  MoveL 9409 to (-39.5, 44.85, 135.08) mm, rotated rx -180 ry 0 rz 180 deg; joints [-167.331, 69.156, -87.298, 166.691, 72.314, 4.11]
  Call Extruder(57.21099)
  MoveL 9410 to (-39.44, 44.66, 135.08) mm, rotated rx 180 ry 0 rz 180 deg; joints [-167.379, 69.148, -87.304, 166.74, 72.298, 4.098]
  MoveL 9411 to (-39.44, 44.66, 135.08) mm, rotated rx 180 ry 0 rz 180 deg; joints [-167.379, 69.148, -87.304, 166.74, 72.298, 4.098]
  Call Extruder(57.35863)
  MoveL 9412 to (-39.35, 44.42, 135.08) mm, rotated rx -180 ry 0 rz 180 deg; joints [-167.439, 69.136, -87.311, 166.802, 72.275, 4.084]
  MoveL 9413 to (-39.35, 44.42, 135.08) mm, rotated rx -180 ry 0 rz 180 deg; joints [-167.439, 69.136, -87.311, 166.802, 72.275, 4.084]
  Call Extruder(57.54097)
  MoveL 9414 to (-39.23, 44.13, 135.08) mm, rotated rx -180 ry 0 rz -180 deg; joints [-167.512, 69.122, -87.32, 166.876, 72.247, 4.066]
  MoveL 9415 to (-39.23, 44.13, 135.08) mm, rotated rx -180 ry 0 rz -180 deg; joints [-167.512, 69.122, -87.32, 166.876, 72.247, 4.066]
  Call Extruder(57.72406)
  MoveL 9416 to (-39.11, 43.83, 135.08) mm, rotated rx 180 ry 0 rz -180 deg; joints [-167.584, 69.107, -87.328, 166.951, 72.219, 4.049]
  MoveL 9417 to (-39.11, 43.83, 135.08) mm, rotated rx 180 ry 0 rz -180 deg; joints [-167.584, 69.107, -87.328, 166.951, 72.219, 4.049]
  Call Extruder(57.88175)
  MoveL 9418 to (-39, 43.58, 135.08) mm, rotated rx -180 ry 0 rz 180 deg; joints [-167.646, 69.094, -87.336, 167.014, 72.194, 4.034]
  MoveL 9419 to (-39, 43.58, 135.08) mm, rotated rx -180 ry 0 rz 180 deg; joints [-167.646, 69.094, -87.336, 167.014, 72.194, 4.034]
  Call Extruder(58.04004)
  MoveL 9420 to (-38.89, 43.33, 135.08) mm, rotated rx 180 ry 0 rz 180 deg; joints [-167.708, 69.081, -87.344, 167.078, 72.17, 4.019]
  MoveL 9421 to (-38.89, 43.33, 135.08) mm, rotated rx 180 ry 0 rz 180 deg; joints [-167.708, 69.081, -87.344, 167.078, 72.17, 4.019]
  Call Extruder(58.22206)
  MoveL 9422 to (-38.75, 43.06, 135.08) mm, rotated rx -180 ry 0 rz 180 deg; joints [-167.776, 69.065, -87.354, 167.147, 72.14, 4.003]
  MoveL 9423 to (-38.75, 43.06, 135.08) mm, rotated rx -180 ry 0 rz 180 deg; joints [-167.776, 69.065, -87.354, 167.147, 72.14, 4.003]
  Call Extruder(58.42862)
  MoveL 9424 to (-38.57, 42.75, 135.08) mm, rotated rx -180 ry 0 rz 180 deg; joints [-167.849, 69.046, -87.365, 167.222, 72.105, 3.986]
  MoveL 9425 to (-38.57, 42.75, 135.08) mm, rotated rx -180 ry 0 rz 180 deg; joints [-167.849, 69.046, -87.365, 167.222, 72.105, 3.986]
  Call Extruder(58.63595)
  MoveL 9426 to (-38.4, 42.45, 135.08) mm, rotated rx -180 ry 0 rz 180 deg; joints [-167.923, 69.027, -87.377, 167.296, 72.07, 3.97]
  MoveL 9427 to (-38.4, 42.45, 135.08) mm, rotated rx -180 ry 0 rz 180 deg; joints [-167.923, 69.027, -87.377, 167.296, 72.07, 3.97]
  Call Extruder(58.84406)
  MoveL 9428 to (-38.22, 42.15, 135.08) mm, rotated rx -180 ry 0 rz 180 deg; joints [-167.997, 69.007, -87.389, 167.371, 72.035, 3.953]
  MoveL 9429 to (-38.22, 42.15, 135.08) mm, rotated rx -180 ry 0 rz 180 deg; joints [-167.997, 69.007, -87.389, 167.371, 72.035, 3.953]
  Call Extruder(58.96178)
  MoveL 9430 to (-38.12, 41.98, 135.08) mm, rotated rx 180 ry 0 rz 180 deg; joints [-168.038, 68.997, -87.395, 167.414, 72.015, 3.944]
  MoveL 9431 to (-38.12, 41.98, 135.08) mm, rotated rx 180 ry 0 rz 180 deg; joints [-168.038, 68.997, -87.395, 167.414, 72.015, 3.944]
  Call Extruder(59.29462)
  MoveL 9432 to (-37.79, 41.52, 135.08) mm, rotated rx -180 ry 0 rz -180 deg; joints [-168.144, 68.962, -87.415, 167.521, 71.955, 3.922]
  MoveL 9433 to (-37.79, 41.52, 135.08) mm, rotated rx -180 ry 0 rz -180 deg; joints [-168.144, 68.962, -87.415, 167.521, 71.955, 3.922]
  Call Extruder(59.62865)
  MoveL 9434 to (-37.47, 41.07, 135.08) mm, rotated rx -180 ry 0 rz 180 deg; joints [-168.25, 68.929, -87.435, 167.629, 71.894, 3.899]
  MoveL 9435 to (-37.47, 41.07, 135.08) mm, rotated rx -180 ry 0 rz 180 deg; joints [-168.25, 68.929, -87.435, 167.629, 71.894, 3.899]
  Call Extruder(59.79624)
  MoveL 9436 to (-37.3, 40.85, 135.08) mm, rotated rx -180 ry 0 rz 180 deg; joints [-168.304, 68.912, -87.445, 167.683, 71.864, 3.888]
  Call Extruder(60.62555)
  MoveL 9437 to (-36.39, 39.81, 135.08) mm, rotated rx 180 ry 0 rz 180 deg; joints [-168.541, 68.821, -87.499, 167.922, 71.708, 3.842]
  Call Extruder(61.25663)
  MoveL 9438 to (-35.6, 39.11, 135.08) mm, rotated rx -180 ry 0 rz 180 deg; joints [-168.693, 68.746, -87.542, 168.074, 71.581, 3.818]
  MoveL 9439 to (-35.6, 39.11, 135.08) mm, rotated rx -180 ry 0 rz 180 deg; joints [-168.693, 68.746, -87.542, 168.074, 71.581, 3.818]
  Call Extruder(61.45419)
  MoveL 9440 to (-35.35, 38.9, 135.08) mm, rotated rx 180 ry 0 rz -180 deg; joints [-168.739, 68.722, -87.556, 168.12, 71.541, 3.811]
  Call Extruder(61.78821)
  MoveL 9441 to (-34.9, 38.57, 135.08) mm, rotated rx 180 ry 0 rz -180 deg; joints [-168.806, 68.68, -87.58, 168.186, 71.472, 3.803]
  MoveL 9442 to (-34.9, 38.57, 135.08) mm, rotated rx 180 ry 0 rz -180 deg; joints [-168.806, 68.68, -87.58, 168.186, 71.472, 3.803]
  Call Extruder(62.12104)
  MoveL 9443 to (-34.45, 38.24, 135.08) mm, rotated rx 180 ry 0 rz 180 deg; joints [-168.874, 68.638, -87.604, 168.253, 71.403, 3.794]
  MoveL 9444 to (-34.45, 38.24, 135.08) mm, rotated rx 180 ry 0 rz 180 deg; joints [-168.874, 68.638, -87.604, 168.253, 71.403, 3.794]
  Call Extruder(62.30029)
  MoveL 9445 to (-34.21, 38.07, 135.08) mm, rotated rx -180 ry 0 rz -180 deg; joints [-168.91, 68.615, -87.617, 168.288, 71.365, 3.79]
  MoveL 9446 to (-34.21, 38.07, 135.08) mm, rotated rx -180 ry 0 rz -180 deg; joints [-168.91, 68.615, -87.617, 168.288, 71.365, 3.79]
  Call Extruder(62.50840)
  MoveL 9447 to (-33.9, 37.89, 135.08) mm, rotated rx 180 ry 0 rz 180 deg; joints [-168.944, 68.587, -87.633, 168.32, 71.321, 3.788]
  MoveL 9448 to (-33.9, 37.89, 135.08) mm, rotated rx 180 ry 0 rz 180 deg; joints [-168.944, 68.587, -87.633, 168.32, 71.321, 3.788]
  Call Extruder(62.71573)
  MoveL 9449 to (-33.6, 37.71, 135.08) mm, rotated rx -180 ry 0 rz -180 deg; joints [-168.977, 68.559, -87.649, 168.352, 71.276, 3.786]
  MoveL 9450 to (-33.6, 37.71, 135.08) mm, rotated rx -180 ry 0 rz -180 deg; joints [-168.977, 68.559, -87.649, 168.352, 71.276, 3.786]
  Call Extruder(62.92229)
  MoveL 9451 to (-33.29, 37.54, 135.08) mm, rotated rx 180 ry 0 rz 180 deg; joints [-169.01, 68.531, -87.664, 168.384, 71.231, 3.784]
  MoveL 9452 to (-33.29, 37.54, 135.08) mm, rotated rx 180 ry 0 rz 180 deg; joints [-169.01, 68.531, -87.664, 168.384, 71.231, 3.784]
  Call Extruder(63.12806)
  MoveL 9453 to (-32.99, 37.36, 135.08) mm, rotated rx 180 ry 0 rz -180 deg; joints [-169.043, 68.504, -87.68, 168.416, 71.187, 3.782]
  MoveL 9454 to (-32.99, 37.36, 135.08) mm, rotated rx 180 ry 0 rz -180 deg; joints [-169.043, 68.504, -87.68, 168.416, 71.187, 3.782]
  Call Extruder(63.28636)
  MoveL 9455 to (-32.74, 37.26, 135.08) mm, rotated rx -180 ry 0 rz 180 deg; joints [-169.06, 68.481, -87.692, 168.432, 71.152, 3.783]
  MoveL 9456 to (-32.74, 37.26, 135.08) mm, rotated rx -180 ry 0 rz 180 deg; joints [-169.06, 68.481, -87.692, 168.432, 71.152, 3.783]
  Call Extruder(63.44406)
  MoveL 9457 to (-32.49, 37.15, 135.08) mm, rotated rx -180 ry 0 rz -180 deg; joints [-169.077, 68.459, -87.704, 168.447, 71.117, 3.785]
  MoveL 9458 to (-32.49, 37.15, 135.08) mm, rotated rx -180 ry 0 rz -180 deg; joints [-169.077, 68.459, -87.704, 168.447, 71.117, 3.785]
  Call Extruder(63.61415)
  MoveL 9459 to (-32.22, 37.04, 135.08) mm, rotated rx -180 ry 0 rz 180 deg; joints [-169.095, 68.435, -87.718, 168.463, 71.079, 3.787]
  MoveL 9460 to (-32.22, 37.04, 135.08) mm, rotated rx -180 ry 0 rz 180 deg; joints [-169.095, 68.435, -87.718, 168.463, 71.079, 3.787]
  Call Extruder(63.79648)
  MoveL 9461 to (-31.93, 36.91, 135.08) mm, rotated rx 180 ry 0 rz 180 deg; joints [-169.113, 68.409, -87.732, 168.48, 71.038, 3.789]
  MoveL 9462 to (-31.93, 36.91, 135.08) mm, rotated rx 180 ry 0 rz 180 deg; joints [-169.113, 68.409, -87.732, 168.48, 71.038, 3.789]
  Call Extruder(63.97805)
  MoveL 9463 to (-31.64, 36.79, 135.08) mm, rotated rx -180 ry 0 rz -180 deg; joints [-169.132, 68.383, -87.746, 168.497, 70.997, 3.791]
  MoveL 9464 to (-31.64, 36.79, 135.08) mm, rotated rx -180 ry 0 rz -180 deg; joints [-169.132, 68.383, -87.746, 168.497, 70.997, 3.791]
  Call Extruder(64.09151)
  MoveL 9465 to (-31.45, 36.73, 135.08) mm, rotated rx -180 ry 0 rz 180 deg; joints [-169.139, 68.366, -87.755, 168.503, 70.972, 3.794]
  MoveL 9466 to (-31.45, 36.73, 135.08) mm, rotated rx -180 ry 0 rz 180 deg; joints [-169.139, 68.366, -87.755, 168.503, 70.972, 3.794]
  Call Extruder(64.20453)
  MoveL 9467 to (-31.26, 36.67, 135.08) mm, rotated rx -180 ry 0 rz -180 deg; joints [-169.146, 68.35, -87.765, 168.509, 70.946, 3.797]
  MoveL 9468 to (-31.26, 36.67, 135.08) mm, rotated rx -180 ry 0 rz -180 deg; joints [-169.146, 68.35, -87.765, 168.509, 70.946, 3.797]
  Call Extruder(64.31709)
  MoveL 9469 to (-31.07, 36.61, 135.08) mm, rotated rx 180 ry 0 rz -180 deg; joints [-169.154, 68.333, -87.774, 168.515, 70.92, 3.8]
  MoveL 9470 to (-31.07, 36.61, 135.08) mm, rotated rx 180 ry 0 rz -180 deg; joints [-169.154, 68.333, -87.774, 168.515, 70.92, 3.8]
  Call Extruder(64.42922)
  MoveL 9471 to (-30.88, 36.55, 135.08) mm, rotated rx -180 ry 0 rz 180 deg; joints [-169.161, 68.316, -87.783, 168.521, 70.895, 3.803]
  MoveL 9472 to (-30.88, 36.55, 135.08) mm, rotated rx -180 ry 0 rz 180 deg; joints [-169.161, 68.316, -87.783, 168.521, 70.895, 3.803]
  Call Extruder(64.54090)
  MoveL 9473 to (-30.69, 36.49, 135.08) mm, rotated rx 180 ry 0 rz 180 deg; joints [-169.168, 68.3, -87.792, 168.527, 70.869, 3.806]
  MoveL 9474 to (-30.69, 36.49, 135.08) mm, rotated rx 180 ry 0 rz 180 deg; joints [-169.168, 68.3, -87.792, 168.527, 70.869, 3.806]
  Call Extruder(64.67197)
  MoveL 9475 to (-30.47, 36.42, 135.08) mm, rotated rx -180 ry 0 rz -180 deg; joints [-169.175, 68.28, -87.802, 168.532, 70.839, 3.809]
  MoveL 9476 to (-30.47, 36.42, 135.08) mm, rotated rx -180 ry 0 rz -180 deg; joints [-169.175, 68.28, -87.802, 168.532, 70.839, 3.809]
  Call Extruder(64.80248)
  MoveL 9477 to (-30.25, 36.35, 135.08) mm, rotated rx -180 ry 0 rz 180 deg; joints [-169.182, 68.26, -87.813, 168.538, 70.809, 3.813]
  MoveL 9478 to (-30.25, 36.35, 135.08) mm, rotated rx -180 ry 0 rz 180 deg; joints [-169.182, 68.26, -87.813, 168.538, 70.809, 3.813]
  Call Extruder(64.93242)
  MoveL 9479 to (-30.02, 36.28, 135.08) mm, rotated rx -180 ry 0 rz -180 deg; joints [-169.19, 68.241, -87.824, 168.543, 70.779, 3.817]
  MoveL 9480 to (-30.02, 36.28, 135.08) mm, rotated rx -180 ry 0 rz -180 deg; joints [-169.19, 68.241, -87.824, 168.543, 70.779, 3.817]
  Call Extruder(65.06180)
  MoveL 9481 to (-29.8, 36.22, 135.08) mm, rotated rx 180 ry 0 rz -180 deg; joints [-169.197, 68.221, -87.834, 168.549, 70.748, 3.821]
  MoveL 9482 to (-29.8, 36.22, 135.08) mm, rotated rx 180 ry 0 rz -180 deg; joints [-169.197, 68.221, -87.834, 168.549, 70.748, 3.821]
  Call Extruder(65.18377)
  MoveL 9483 to (-29.59, 36.16, 135.08) mm, rotated rx -180 ry 0 rz 180 deg; joints [-169.202, 68.202, -87.844, 168.552, 70.72, 3.826]
  MoveL 9484 to (-29.59, 36.16, 135.08) mm, rotated rx -180 ry 0 rz 180 deg; joints [-169.202, 68.202, -87.844, 168.552, 70.72, 3.826]
  Call Extruder(65.29861)
  MoveL 9485 to (-29.38, 36.12, 135.08) mm, rotated rx -180 ry 0 rz 180 deg; joints [-169.203, 68.185, -87.854, 168.551, 70.693, 3.831]
  MoveL 9486 to (-29.38, 36.12, 135.08) mm, rotated rx -180 ry 0 rz 180 deg; joints [-169.203, 68.185, -87.854, 168.551, 70.693, 3.831]
  Call Extruder(65.41301)
  MoveL 9487 to (-29.18, 36.07, 135.08) mm, rotated rx -180 ry 0 rz 180 deg; joints [-169.205, 68.167, -87.863, 168.551, 70.666, 3.836]
  MoveL 9488 to (-29.18, 36.07, 135.08) mm, rotated rx -180 ry 0 rz 180 deg; joints [-169.205, 68.167, -87.863, 168.551, 70.666, 3.836]
  Call Extruder(65.52695)
  MoveL 9489 to (-28.97, 36.03, 135.08) mm, rotated rx -180 ry 0 rz -180 deg; joints [-169.207, 68.149, -87.872, 168.551, 70.64, 3.841]
  MoveL 9490 to (-28.97, 36.03, 135.08) mm, rotated rx -180 ry 0 rz -180 deg; joints [-169.207, 68.149, -87.872, 168.551, 70.64, 3.841]
  Call Extruder(65.64044)
  MoveL 9491 to (-28.77, 35.98, 135.08) mm, rotated rx 180 ry 0 rz 180 deg; joints [-169.208, 68.131, -87.882, 168.551, 70.613, 3.846]
  MoveL 9492 to (-28.77, 35.98, 135.08) mm, rotated rx 180 ry 0 rz 180 deg; joints [-169.208, 68.131, -87.882, 168.551, 70.613, 3.846]
  Call Extruder(65.77772)
  MoveL 9493 to (-28.52, 35.93, 135.08) mm, rotated rx -180 ry 0 rz -180 deg; joints [-169.209, 68.11, -87.893, 168.549, 70.58, 3.853]
  MoveL 9494 to (-28.52, 35.93, 135.08) mm, rotated rx -180 ry 0 rz -180 deg; joints [-169.209, 68.11, -87.893, 168.549, 70.58, 3.853]
  Call Extruder(65.91440)
  MoveL 9495 to (-28.27, 35.88, 135.08) mm, rotated rx -180 ry 0 rz 180 deg; joints [-169.209, 68.088, -87.905, 168.547, 70.548, 3.86]
  MoveL 9496 to (-28.27, 35.88, 135.08) mm, rotated rx -180 ry 0 rz 180 deg; joints [-169.209, 68.088, -87.905, 168.547, 70.548, 3.86]
  Call Extruder(66.05046)
  MoveL 9497 to (-28.02, 35.83, 135.08) mm, rotated rx -180 ry 0 rz 180 deg; joints [-169.21, 68.066, -87.916, 168.546, 70.515, 3.866]
  MoveL 9498 to (-28.02, 35.83, 135.08) mm, rotated rx -180 ry 0 rz 180 deg; joints [-169.21, 68.066, -87.916, 168.546, 70.515, 3.866]
  Call Extruder(66.18591)
  MoveL 9499 to (-27.77, 35.78, 135.08) mm, rotated rx 180 ry 0 rz 180 deg; joints [-169.21, 68.044, -87.928, 168.544, 70.483, 3.873]
  MoveL 9500 to (-27.77, 35.78, 135.08) mm, rotated rx 180 ry 0 rz 180 deg; joints [-169.21, 68.044, -87.928, 168.544, 70.483, 3.873]
  Call Extruder(66.32075)
  MoveL 9501 to (-27.52, 35.73, 135.08) mm, rotated rx 180 ry 0 rz 180 deg; joints [-169.211, 68.023, -87.939, 168.543, 70.45, 3.88]
  MoveL 9502 to (-27.52, 35.73, 135.08) mm, rotated rx 180 ry 0 rz 180 deg; joints [-169.211, 68.023, -87.939, 168.543, 70.45, 3.88]
  Call Extruder(66.45498)
  MoveL 9503 to (-27.28, 35.68, 135.08) mm, rotated rx -180 ry 0 rz 180 deg; joints [-169.212, 68.001, -87.95, 168.541, 70.418, 3.887]
  MoveL 9504 to (-27.28, 35.68, 135.08) mm, rotated rx -180 ry 0 rz 180 deg; joints [-169.212, 68.001, -87.95, 168.541, 70.418, 3.887]
  Call Extruder(66.58860)
  MoveL 9505 to (-27.03, 35.63, 135.08) mm, rotated rx -180 ry 0 rz 180 deg; joints [-169.212, 67.979, -87.961, 168.539, 70.386, 3.893]
  MoveL 9506 to (-27.03, 35.63, 135.08) mm, rotated rx -180 ry 0 rz 180 deg; joints [-169.212, 67.979, -87.961, 168.539, 70.386, 3.893]
  Call Extruder(66.75070)
  MoveL 9507 to (-26.72, 35.59, 135.08) mm, rotated rx -180 ry 0 rz -180 deg; joints [-169.21, 67.953, -87.975, 168.533, 70.346, 3.903]
  MoveL 9508 to (-26.72, 35.59, 135.08) mm, rotated rx -180 ry 0 rz -180 deg; joints [-169.21, 67.953, -87.975, 168.533, 70.346, 3.903]
  Call Extruder(66.91207)
  MoveL 9509 to (-26.41, 35.54, 135.08) mm, rotated rx 180 ry 0 rz 180 deg; joints [-169.207, 67.926, -87.989, 168.527, 70.307, 3.913]
  MoveL 9510 to (-26.41, 35.54, 135.08) mm, rotated rx 180 ry 0 rz 180 deg; joints [-169.207, 67.926, -87.989, 168.527, 70.307, 3.913]
  Call Extruder(67.07271)
  MoveL 9511 to (-26.11, 35.49, 135.08) mm, rotated rx -180 ry 0 rz -180 deg; joints [-169.204, 67.899, -88.003, 168.521, 70.268, 3.922]
  MoveL 9512 to (-26.11, 35.49, 135.08) mm, rotated rx -180 ry 0 rz -180 deg; joints [-169.204, 67.899, -88.003, 168.521, 70.268, 3.922]
  Call Extruder(67.23263)
  MoveL 9513 to (-25.8, 35.44, 135.08) mm, rotated rx -180 ry 0 rz 180 deg; joints [-169.201, 67.873, -88.016, 168.515, 70.228, 3.932]
  MoveL 9514 to (-25.8, 35.44, 135.08) mm, rotated rx -180 ry 0 rz 180 deg; joints [-169.201, 67.873, -88.016, 168.515, 70.228, 3.932]
  Call Extruder(67.39181)
  MoveL 9515 to (-25.5, 35.39, 135.08) mm, rotated rx -180 ry 0 rz 180 deg; joints [-169.198, 67.846, -88.03, 168.51, 70.189, 3.941]
  MoveL 9516 to (-25.5, 35.39, 135.08) mm, rotated rx -180 ry 0 rz 180 deg; joints [-169.198, 67.846, -88.03, 168.51, 70.189, 3.941]
  Call Extruder(67.55027)
  MoveL 9517 to (-25.19, 35.34, 135.08) mm, rotated rx -180 ry 0 rz 180 deg; joints [-169.195, 67.819, -88.043, 168.503, 70.15, 3.951]
  MoveL 9518 to (-25.19, 35.34, 135.08) mm, rotated rx -180 ry 0 rz 180 deg; joints [-169.195, 67.819, -88.043, 168.503, 70.15, 3.951]
  Call Extruder(67.74915)
  MoveL 9519 to (-24.8, 35.3, 135.08) mm, rotated rx -180 ry 0 rz 180 deg; joints [-169.187, 67.786, -88.06, 168.491, 70.101, 3.965]
  MoveL 9520 to (-24.8, 35.3, 135.08) mm, rotated rx -180 ry 0 rz 180 deg; joints [-169.187, 67.786, -88.06, 168.491, 70.101, 3.965]
  Call Extruder(67.94716)
  MoveL 9521 to (-24.42, 35.25, 135.08) mm, rotated rx -180 ry 0 rz -180 deg; joints [-169.178, 67.752, -88.077, 168.478, 70.052, 3.978]
  MoveL 9522 to (-24.42, 35.25, 135.08) mm, rotated rx -180 ry 0 rz -180 deg; joints [-169.178, 67.752, -88.077, 168.478, 70.052, 3.978]
  Call Extruder(68.14430)
  MoveL 9523 to (-24.03, 35.21, 135.08) mm, rotated rx 180 ry 0 rz -180 deg; joints [-169.17, 67.718, -88.094, 168.466, 70.003, 3.992]
  MoveL 9524 to (-24.03, 35.21, 135.08) mm, rotated rx 180 ry 0 rz -180 deg; joints [-169.17, 67.718, -88.094, 168.466, 70.003, 3.992]
  Call Extruder(68.34057)
  MoveL 9525 to (-23.64, 35.16, 135.08) mm, rotated rx -180 ry 0 rz -180 deg; joints [-169.161, 67.684, -88.111, 168.453, 69.954, 4.006]
  MoveL 9526 to (-23.64, 35.16, 135.08) mm, rotated rx -180 ry 0 rz -180 deg; joints [-169.161, 67.684, -88.111, 168.453, 69.954, 4.006]
  Call Extruder(68.58626)
  MoveL 9527 to (-23.15, 35.11, 135.08) mm, rotated rx -180 ry 0 rz 180 deg; joints [-169.147, 67.642, -88.132, 168.433, 69.893, 4.025]
  MoveL 9528 to (-23.15, 35.11, 135.08) mm, rotated rx -180 ry 0 rz 180 deg; joints [-169.147, 67.642, -88.132, 168.433, 69.893, 4.025]
  Call Extruder(68.88099)
  MoveL 9529 to (-22.56, 35.07, 135.08) mm, rotated rx 180 ry 0 rz 180 deg; joints [-169.127, 67.591, -88.157, 168.406, 69.819, 4.048]
  MoveL 9530 to (-22.56, 35.07, 135.08) mm, rotated rx 180 ry 0 rz 180 deg; joints [-169.127, 67.591, -88.157, 168.406, 69.819, 4.048]
  Call Extruder(69.17439)
  MoveL 9531 to (-21.97, 35.02, 135.08) mm, rotated rx -180 ry 0 rz 180 deg; joints [-169.107, 67.539, -88.182, 168.379, 69.746, 4.072]
  MoveL 9532 to (-21.97, 35.02, 135.08) mm, rotated rx -180 ry 0 rz 180 deg; joints [-169.107, 67.539, -88.182, 168.379, 69.746, 4.072]
  Call Extruder(69.60772)
  MoveL 9533 to (-21.1, 34.98, 135.08) mm, rotated rx 180 ry 0 rz -180 deg; joints [-169.069, 67.463, -88.219, 168.331, 69.638, 4.11]
  MoveL 9534 to (-21.1, 34.98, 135.08) mm, rotated rx 180 ry 0 rz -180 deg; joints [-169.069, 67.463, -88.219, 168.331, 69.638, 4.11]
  Call Extruder(70.17988)
  MoveL 9535 to (-19.94, 34.93, 135.08) mm, rotated rx -180 ry 0 rz -180 deg; joints [-169.014, 67.362, -88.267, 168.261, 69.496, 4.163]
  MoveL 9536 to (-19.94, 34.93, 135.08) mm, rotated rx -180 ry 0 rz -180 deg; joints [-169.014, 67.362, -88.267, 168.261, 69.496, 4.163]
  Call Extruder(70.60771)
  MoveL 9537 to (-19.06, 34.91, 135.08) mm, rotated rx -180 ry 0 rz -180 deg; joints [-168.967, 67.286, -88.303, 168.202, 69.39, 4.205]
  Call Extruder(187.25639)
  MoveL 9538 to (219.06, 34.91, 135.08) mm, rotated rx 180 ry 0 rz -180 deg; joints [-30.588, 55.377, -90.527, 35.864, 119.71, 19.712]
  MoveL 9539 to (219.06, 34.91, 135.08) mm, rotated rx 180 ry 0 rz -180 deg; joints [-30.588, 55.377, -90.527, 35.864, 119.71, 19.712]
  Call Extruder(187.97196)
  MoveL 9540 to (220.52, 34.95, 135.08) mm, rotated rx -180 ry 0 rz 180 deg; joints [-30.009, 55.529, -90.53, 35.187, 119.782, 19.301]
  MoveL 9541 to (220.52, 34.95, 135.08) mm, rotated rx -180 ry 0 rz 180 deg; joints [-30.009, 55.529, -90.53, 35.187, 119.782, 19.301]
  Call Extruder(188.54670)
  MoveL 9542 to (221.68, 35, 135.08) mm, rotated rx 180 ry 0 rz 180 deg; joints [-29.572, 55.651, -90.532, 34.671, 119.826, 18.984]
  MoveL 9543 to (221.68, 35, 135.08) mm, rotated rx 180 ry 0 rz 180 deg; joints [-29.572, 55.651, -90.532, 34.671, 119.826, 18.984]
  Call Extruder(188.84009)
  MoveL 9544 to (222.27, 35.04, 135.08) mm, rotated rx -180 ry 0 rz 180 deg; joints [-29.371, 55.715, -90.532, 34.432, 119.839, 18.834]
  MoveL 9545 to (222.27, 35.04, 135.08) mm, rotated rx -180 ry 0 rz 180 deg; joints [-29.371, 55.715, -90.532, 34.432, 119.839, 18.834]
  Call Extruder(189.13482)
  MoveL 9546 to (222.86, 35.09, 135.08) mm, rotated rx -180 ry 0 rz 180 deg; joints [-29.173, 55.779, -90.533, 34.195, 119.851, 18.686]
  MoveL 9547 to (222.86, 35.09, 135.08) mm, rotated rx -180 ry 0 rz 180 deg; joints [-29.173, 55.779, -90.533, 34.195, 119.851, 18.686]
  Call Extruder(189.43087)
  MoveL 9548 to (223.45, 35.14, 135.08) mm, rotated rx -180 ry 0 rz -180 deg; joints [-28.978, 55.842, -90.534, 33.962, 119.861, 18.539]
  MoveL 9549 to (223.45, 35.14, 135.08) mm, rotated rx -180 ry 0 rz -180 deg; joints [-28.978, 55.842, -90.534, 33.962, 119.861, 18.539]
  Call Extruder(189.62715)
  MoveL 9550 to (223.84, 35.18, 135.08) mm, rotated rx 180 ry 0 rz 180 deg; joints [-28.862, 55.885, -90.534, 33.821, 119.863, 18.449]
  MoveL 9551 to (223.84, 35.18, 135.08) mm, rotated rx 180 ry 0 rz 180 deg; joints [-28.862, 55.885, -90.534, 33.821, 119.863, 18.449]
  Call Extruder(189.82429)
  MoveL 9552 to (224.22, 35.23, 135.08) mm, rotated rx 180 ry 0 rz 180 deg; joints [-28.747, 55.928, -90.534, 33.682, 119.864, 18.359]
  MoveL 9553 to (224.22, 35.23, 135.08) mm, rotated rx 180 ry 0 rz 180 deg; joints [-28.747, 55.928, -90.534, 33.682, 119.864, 18.359]
  Call Extruder(190.02230)
  MoveL 9554 to (224.61, 35.28, 135.08) mm, rotated rx 180 ry 0 rz -180 deg; joints [-28.633, 55.97, -90.534, 33.544, 119.864, 18.27]
  MoveL 9555 to (224.61, 35.28, 135.08) mm, rotated rx 180 ry 0 rz -180 deg; joints [-28.633, 55.97, -90.534, 33.544, 119.864, 18.27]
  Call Extruder(190.22117)
  MoveL 9556 to (225, 35.32, 135.08) mm, rotated rx -180 ry 0 rz 180 deg; joints [-28.52, 56.013, -90.535, 33.407, 119.864, 18.181]
  MoveL 9557 to (225, 35.32, 135.08) mm, rotated rx -180 ry 0 rz 180 deg; joints [-28.52, 56.013, -90.535, 33.407, 119.864, 18.181]
  Call Extruder(190.40025)
  MoveL 9558 to (225.34, 35.37, 135.08) mm, rotated rx -180 ry 0 rz 180 deg; joints [-28.425, 56.052, -90.535, 33.29, 119.862, 18.105]
  MoveL 9559 to (225.34, 35.37, 135.08) mm, rotated rx -180 ry 0 rz 180 deg; joints [-28.425, 56.052, -90.535, 33.29, 119.862, 18.105]
  Call Extruder(190.55944)
  MoveL 9560 to (225.65, 35.42, 135.08) mm, rotated rx -180 ry 0 rz 180 deg; joints [-28.346, 56.086, -90.535, 33.193, 119.857, 18.04]
  MoveL 9561 to (225.65, 35.42, 135.08) mm, rotated rx -180 ry 0 rz 180 deg; joints [-28.346, 56.086, -90.535, 33.193, 119.857, 18.04]
  Call Extruder(190.71935)
  MoveL 9562 to (225.96, 35.47, 135.08) mm, rotated rx 180 ry 0 rz 180 deg; joints [-28.267, 56.121, -90.535, 33.096, 119.853, 17.975]
  MoveL 9563 to (225.96, 35.47, 135.08) mm, rotated rx 180 ry 0 rz 180 deg; joints [-28.267, 56.121, -90.535, 33.096, 119.853, 17.975]
  Call Extruder(190.87999)
  MoveL 9564 to (226.26, 35.51, 135.08) mm, rotated rx -180 ry 0 rz 180 deg; joints [-28.19, 56.155, -90.535, 33, 119.848, 17.911]
  MoveL 9565 to (226.26, 35.51, 135.08) mm, rotated rx -180 ry 0 rz 180 deg; joints [-28.19, 56.155, -90.535, 33, 119.848, 17.911]
  Call Extruder(191.04136)
  MoveL 9566 to (226.57, 35.56, 135.08) mm, rotated rx 180 ry 0 rz 180 deg; joints [-28.112, 56.189, -90.535, 32.904, 119.843, 17.847]
  MoveL 9567 to (226.57, 35.56, 135.08) mm, rotated rx 180 ry 0 rz 180 deg; joints [-28.112, 56.189, -90.535, 32.904, 119.843, 17.847]
  Call Extruder(191.20345)
  MoveL 9568 to (226.87, 35.61, 135.08) mm, rotated rx 180 ry 0 rz 180 deg; joints [-28.036, 56.224, -90.535, 32.81, 119.837, 17.784]
  MoveL 9569 to (226.87, 35.61, 135.08) mm, rotated rx 180 ry 0 rz 180 deg; joints [-28.036, 56.224, -90.535, 32.81, 119.837, 17.784]
  Call Extruder(191.35165)
  MoveL 9570 to (227.15, 35.66, 135.08) mm, rotated rx -180 ry 0 rz -180 deg; joints [-27.971, 56.255, -90.535, 32.728, 119.83, 17.729]
  MoveL 9571 to (227.15, 35.66, 135.08) mm, rotated rx -180 ry 0 rz -180 deg; joints [-27.971, 56.255, -90.535, 32.728, 119.83, 17.729]
  Call Extruder(191.48588)
  MoveL 9572 to (227.4, 35.71, 135.08) mm, rotated rx -180 ry 0 rz 180 deg; joints [-27.915, 56.284, -90.534, 32.659, 119.823, 17.681]
  MoveL 9573 to (227.4, 35.71, 135.08) mm, rotated rx -180 ry 0 rz 180 deg; joints [-27.915, 56.284, -90.534, 32.659, 119.823, 17.681]
  Call Extruder(191.62072)
  MoveL 9574 to (227.65, 35.76, 135.08) mm, rotated rx -180 ry 0 rz 180 deg; joints [-27.861, 56.312, -90.534, 32.59, 119.815, 17.633]
  MoveL 9575 to (227.65, 35.76, 135.08) mm, rotated rx -180 ry 0 rz 180 deg; joints [-27.861, 56.312, -90.534, 32.59, 119.815, 17.633]
  Call Extruder(191.75618)
  MoveL 9576 to (227.9, 35.81, 135.08) mm, rotated rx -180 ry 0 rz 180 deg; joints [-27.807, 56.341, -90.534, 32.521, 119.808, 17.586]
  MoveL 9577 to (227.9, 35.81, 135.08) mm, rotated rx -180 ry 0 rz 180 deg; joints [-27.807, 56.341, -90.534, 32.521, 119.808, 17.586]
  Call Extruder(191.89224)
  MoveL 9578 to (228.15, 35.86, 135.08) mm, rotated rx -180 ry 0 rz 180 deg; joints [-27.753, 56.37, -90.534, 32.454, 119.8, 17.539]
  MoveL 9579 to (228.15, 35.86, 135.08) mm, rotated rx -180 ry 0 rz 180 deg; joints [-27.753, 56.37, -90.534, 32.454, 119.8, 17.539]
  Call Extruder(192.02891)
  MoveL 9580 to (228.4, 35.91, 135.08) mm, rotated rx -180 ry 0 rz -180 deg; joints [-27.699, 56.398, -90.534, 32.385, 119.792, 17.491]
  MoveL 9581 to (228.4, 35.91, 135.08) mm, rotated rx -180 ry 0 rz -180 deg; joints [-27.699, 56.398, -90.534, 32.385, 119.792, 17.491]
  Call Extruder(192.16620)
  MoveL 9582 to (228.65, 35.96, 135.08) mm, rotated rx 180 ry 0 rz 180 deg; joints [-27.646, 56.427, -90.534, 32.319, 119.783, 17.445]
  MoveL 9583 to (228.65, 35.96, 135.08) mm, rotated rx 180 ry 0 rz 180 deg; joints [-27.646, 56.427, -90.534, 32.319, 119.783, 17.445]
  Call Extruder(192.29187)
  MoveL 9584 to (228.87, 36, 135.08) mm, rotated rx -180 ry 0 rz -180 deg; joints [-27.599, 56.453, -90.533, 32.259, 119.775, 17.403]
  MoveL 9585 to (228.87, 36, 135.08) mm, rotated rx -180 ry 0 rz -180 deg; joints [-27.599, 56.453, -90.533, 32.259, 119.775, 17.403]
  Call Extruder(192.40582)
  MoveL 9586 to (229.08, 36.05, 135.08) mm, rotated rx -180 ry 0 rz 180 deg; joints [-27.559, 56.476, -90.533, 32.207, 119.767, 17.366]
  MoveL 9587 to (229.08, 36.05, 135.08) mm, rotated rx -180 ry 0 rz 180 deg; joints [-27.559, 56.476, -90.533, 32.207, 119.767, 17.366]
  Call Extruder(192.52022)
  MoveL 9588 to (229.28, 36.09, 135.08) mm, rotated rx 180 ry 0 rz 180 deg; joints [-27.518, 56.5, -90.533, 32.156, 119.759, 17.33]
  MoveL 9589 to (229.28, 36.09, 135.08) mm, rotated rx 180 ry 0 rz 180 deg; joints [-27.518, 56.5, -90.533, 32.156, 119.759, 17.33]
  Call Extruder(192.63507)
  MoveL 9590 to (229.48, 36.14, 135.08) mm, rotated rx -180 ry 0 rz -180 deg; joints [-27.479, 56.524, -90.533, 32.105, 119.75, 17.293]
  MoveL 9591 to (229.48, 36.14, 135.08) mm, rotated rx -180 ry 0 rz -180 deg; joints [-27.479, 56.524, -90.533, 32.105, 119.75, 17.293]
  Call Extruder(192.75038)
  MoveL 9592 to (229.69, 36.18, 135.08) mm, rotated rx 180 ry 0 rz 180 deg; joints [-27.439, 56.547, -90.532, 32.054, 119.742, 17.257]
  MoveL 9593 to (229.69, 36.18, 135.08) mm, rotated rx 180 ry 0 rz 180 deg; joints [-27.439, 56.547, -90.532, 32.054, 119.742, 17.257]
  Call Extruder(192.82364)
  MoveL 9594 to (229.82, 36.22, 135.08) mm, rotated rx -180 ry 0 rz 180 deg; joints [-27.421, 56.562, -90.532, 32.029, 119.734, 17.238]
  MoveL 9595 to (229.82, 36.22, 135.08) mm, rotated rx -180 ry 0 rz 180 deg; joints [-27.421, 56.562, -90.532, 32.029, 119.734, 17.238]
  Call Extruder(192.95114)
  MoveL 9596 to (230.03, 36.29, 135.08) mm, rotated rx -180 ry 0 rz 180 deg; joints [-27.39, 56.589, -90.532, 31.987, 119.721, 17.205]
  MoveL 9597 to (230.03, 36.29, 135.08) mm, rotated rx -180 ry 0 rz 180 deg; joints [-27.39, 56.589, -90.532, 31.987, 119.721, 17.205]
  Call Extruder(193.07920)
  MoveL 9598 to (230.25, 36.35, 135.08) mm, rotated rx -180 ry 0 rz 180 deg; joints [-27.36, 56.615, -90.532, 31.946, 119.707, 17.172]
  MoveL 9599 to (230.25, 36.35, 135.08) mm, rotated rx -180 ry 0 rz 180 deg; joints [-27.36, 56.615, -90.532, 31.946, 119.707, 17.172]
  Call Extruder(193.20780)
  MoveL 9600 to (230.48, 36.42, 135.08) mm, rotated rx 180 ry 0 rz -180 deg; joints [-27.329, 56.642, -90.531, 31.904, 119.693, 17.139]
  MoveL 9601 to (230.48, 36.42, 135.08) mm, rotated rx 180 ry 0 rz -180 deg; joints [-27.329, 56.642, -90.531, 31.904, 119.693, 17.139]
  Call Extruder(193.33694)
  MoveL 9602 to (230.7, 36.49, 135.08) mm, rotated rx -180 ry 0 rz -180 deg; joints [-27.299, 56.668, -90.531, 31.863, 119.679, 17.106]
  MoveL 9603 to (230.7, 36.49, 135.08) mm, rotated rx -180 ry 0 rz -180 deg; joints [-27.299, 56.668, -90.531, 31.863, 119.679, 17.106]
  Call Extruder(193.44884)
  MoveL 9604 to (230.88, 36.55, 135.08) mm, rotated rx 180 ry 0 rz -180 deg; joints [-27.276, 56.691, -90.53, 31.831, 119.667, 17.08]
  MoveL 9605 to (230.88, 36.55, 135.08) mm, rotated rx 180 ry 0 rz -180 deg; joints [-27.276, 56.691, -90.53, 31.831, 119.667, 17.08]
  Call Extruder(193.56118)
  MoveL 9606 to (231.07, 36.61, 135.08) mm, rotated rx 180 ry 0 rz 180 deg; joints [-27.253, 56.714, -90.53, 31.798, 119.654, 17.053]
  MoveL 9607 to (231.07, 36.61, 135.08) mm, rotated rx 180 ry 0 rz 180 deg; joints [-27.253, 56.714, -90.53, 31.798, 119.654, 17.053]
  Call Extruder(193.67397)
  MoveL 9608 to (231.26, 36.67, 135.08) mm, rotated rx -180 ry 0 rz -180 deg; joints [-27.231, 56.736, -90.53, 31.767, 119.64, 17.027]
  MoveL 9609 to (231.26, 36.67, 135.08) mm, rotated rx -180 ry 0 rz -180 deg; joints [-27.231, 56.736, -90.53, 31.767, 119.64, 17.027]
  Call Extruder(193.78720)
  MoveL 9610 to (231.45, 36.73, 135.08) mm, rotated rx 180 ry 0 rz 180 deg; joints [-27.208, 56.759, -90.529, 31.735, 119.627, 17]
  MoveL 9611 to (231.45, 36.73, 135.08) mm, rotated rx 180 ry 0 rz 180 deg; joints [-27.208, 56.759, -90.529, 31.735, 119.627, 17]
  Call Extruder(193.90088)
  MoveL 9612 to (231.64, 36.79, 135.08) mm, rotated rx -180 ry 0 rz -180 deg; joints [-27.185, 56.782, -90.529, 31.703, 119.614, 16.974]
  MoveL 9613 to (231.64, 36.79, 135.08) mm, rotated rx -180 ry 0 rz -180 deg; joints [-27.185, 56.782, -90.529, 31.703, 119.614, 16.974]
  Call Extruder(194.08284)
  MoveL 9614 to (231.93, 36.91, 135.08) mm, rotated rx -180 ry 0 rz -180 deg; joints [-27.167, 56.819, -90.528, 31.672, 119.588, 16.941]
  MoveL 9615 to (231.93, 36.91, 135.08) mm, rotated rx -180 ry 0 rz -180 deg; joints [-27.167, 56.819, -90.528, 31.672, 119.588, 16.941]
  Call Extruder(194.26556)
  MoveL 9616 to (232.22, 37.04, 135.08) mm, rotated rx 180 ry 0 rz 180 deg; joints [-27.149, 56.855, -90.527, 31.641, 119.561, 16.909]
  MoveL 9617 to (232.22, 37.04, 135.08) mm, rotated rx 180 ry 0 rz 180 deg; joints [-27.149, 56.855, -90.527, 31.641, 119.561, 16.909]
  Call Extruder(194.43598)
  MoveL 9618 to (232.49, 37.15, 135.08) mm, rotated rx -180 ry 0 rz -180 deg; joints [-27.133, 56.889, -90.527, 31.613, 119.536, 16.88]
  MoveL 9619 to (232.49, 37.15, 135.08) mm, rotated rx -180 ry 0 rz -180 deg; joints [-27.133, 56.889, -90.527, 31.613, 119.536, 16.88]
  Call Extruder(194.59398)
  MoveL 9620 to (232.74, 37.26, 135.08) mm, rotated rx 180 ry 0 rz 180 deg; joints [-27.121, 56.921, -90.526, 31.59, 119.513, 16.854]
  MoveL 9621 to (232.74, 37.26, 135.08) mm, rotated rx 180 ry 0 rz 180 deg; joints [-27.121, 56.921, -90.526, 31.59, 119.513, 16.854]
  Call Extruder(194.75258)
  MoveL 9622 to (232.99, 37.36, 135.08) mm, rotated rx 180 ry 0 rz 180 deg; joints [-27.108, 56.952, -90.525, 31.566, 119.489, 16.827]
  MoveL 9623 to (232.99, 37.36, 135.08) mm, rotated rx 180 ry 0 rz 180 deg; joints [-27.108, 56.952, -90.525, 31.566, 119.489, 16.827]
  Call Extruder(194.95874)
  MoveL 9624 to (233.29, 37.54, 135.08) mm, rotated rx 180 ry 0 rz 180 deg; joints [-27.12, 56.993, -90.524, 31.567, 119.45, 16.809]
  MoveL 9625 to (233.29, 37.54, 135.08) mm, rotated rx 180 ry 0 rz 180 deg; joints [-27.12, 56.993, -90.524, 31.567, 119.45, 16.809]
  Call Extruder(195.16569)
  MoveL 9626 to (233.6, 37.71, 135.08) mm, rotated rx -180 ry 0 rz 180 deg; joints [-27.132, 57.034, -90.523, 31.568, 119.411, 16.79]
  MoveL 9627 to (233.6, 37.71, 135.08) mm, rotated rx -180 ry 0 rz 180 deg; joints [-27.132, 57.034, -90.523, 31.568, 119.411, 16.79]
  Call Extruder(195.37341)
  MoveL 9628 to (233.9, 37.89, 135.08) mm, rotated rx 180 ry 0 rz 180 deg; joints [-27.144, 57.074, -90.522, 31.569, 119.372, 16.772]
  MoveL 9629 to (233.9, 37.89, 135.08) mm, rotated rx 180 ry 0 rz 180 deg; joints [-27.144, 57.074, -90.522, 31.569, 119.372, 16.772]
  Call Extruder(195.58192)
  MoveL 9630 to (234.21, 38.07, 135.08) mm, rotated rx -180 ry 0 rz 180 deg; joints [-27.156, 57.115, -90.521, 31.57, 119.333, 16.753]
  MoveL 9631 to (234.21, 38.07, 135.08) mm, rotated rx -180 ry 0 rz 180 deg; joints [-27.156, 57.115, -90.521, 31.57, 119.333, 16.753]
  Call Extruder(195.76146)
  MoveL 9632 to (234.45, 38.24, 135.08) mm, rotated rx -180 ry 0 rz 180 deg; joints [-27.187, 57.149, -90.52, 31.593, 119.294, 16.748]
  MoveL 9633 to (234.45, 38.24, 135.08) mm, rotated rx -180 ry 0 rz 180 deg; joints [-27.187, 57.149, -90.52, 31.593, 119.294, 16.748]
  Call Extruder(196.09487)
  MoveL 9634 to (234.9, 38.57, 135.08) mm, rotated rx 180 ry 0 rz 180 deg; joints [-27.245, 57.213, -90.518, 31.638, 119.221, 16.74]
  MoveL 9635 to (234.9, 38.57, 135.08) mm, rotated rx 180 ry 0 rz 180 deg; joints [-27.245, 57.213, -90.518, 31.638, 119.221, 16.74]
  Call Extruder(196.42947)
  MoveL 9636 to (235.35, 38.9, 135.08) mm, rotated rx 180 ry 0 rz 180 deg; joints [-27.302, 57.277, -90.516, 31.681, 119.148, 16.731]
  Call Extruder(197.25742)
  MoveL 9637 to (236.39, 39.81, 135.08) mm, rotated rx -180 ry 0 rz -180 deg; joints [-27.525, 57.431, -90.511, 31.879, 118.948, 16.753]
  Call Extruder(198.08537)
  MoveL 9638 to (237.3, 40.85, 135.08) mm, rotated rx -180 ry 0 rz 180 deg; joints [-27.851, 57.58, -90.505, 32.19, 118.723, 16.832]
  Call Extruder(198.25267)
  MoveL 9639 to (237.47, 41.07, 135.08) mm, rotated rx -180 ry 0 rz 180 deg; joints [-27.932, 57.608, -90.504, 32.269, 118.675, 16.856]
  MoveL 9640 to (237.47, 41.07, 135.08) mm, rotated rx -180 ry 0 rz 180 deg; joints [-27.932, 57.608, -90.504, 32.269, 118.675, 16.856]
  Call Extruder(198.58609)
  MoveL 9641 to (237.79, 41.52, 135.08) mm, rotated rx -180 ry 0 rz -180 deg; joints [-28.091, 57.666, -90.501, 32.425, 118.578, 16.902]
  MoveL 9642 to (237.79, 41.52, 135.08) mm, rotated rx -180 ry 0 rz -180 deg; joints [-28.091, 57.666, -90.501, 32.425, 118.578, 16.902]
  Call Extruder(198.91833)
  MoveL 9643 to (238.12, 41.97, 135.08) mm, rotated rx -180 ry 0 rz 180 deg; joints [-28.249, 57.724, -90.498, 32.579, 118.481, 16.947]
  MoveL 9644 to (238.12, 41.97, 135.08) mm, rotated rx -180 ry 0 rz 180 deg; joints [-28.249, 57.724, -90.498, 32.579, 118.481, 16.947]
  Call Extruder(199.03601)
  MoveL 9645 to (238.22, 42.15, 135.08) mm, rotated rx 180 ry 0 rz 180 deg; joints [-28.315, 57.743, -90.497, 32.646, 118.444, 16.97]
  MoveL 9646 to (238.22, 42.15, 135.08) mm, rotated rx 180 ry 0 rz 180 deg; joints [-28.315, 57.743, -90.497, 32.646, 118.444, 16.97]
  Call Extruder(199.24373)
  MoveL 9647 to (238.4, 42.45, 135.08) mm, rotated rx 180 ry 0 rz 180 deg; joints [-28.434, 57.777, -90.496, 32.764, 118.38, 17.009]
  MoveL 9648 to (238.4, 42.45, 135.08) mm, rotated rx 180 ry 0 rz 180 deg; joints [-28.434, 57.777, -90.496, 32.764, 118.38, 17.009]
  Call Extruder(199.45067)
  MoveL 9649 to (238.57, 42.75, 135.08) mm, rotated rx 180 ry 0 rz -180 deg; joints [-28.552, 57.811, -90.494, 32.882, 118.315, 17.048]
  MoveL 9650 to (238.57, 42.75, 135.08) mm, rotated rx 180 ry 0 rz -180 deg; joints [-28.552, 57.811, -90.494, 32.882, 118.315, 17.048]
  Call Extruder(199.65683)
  MoveL 9651 to (238.75, 43.06, 135.08) mm, rotated rx -180 ry 0 rz 180 deg; joints [-28.669, 57.845, -90.493, 32.998, 118.251, 17.086]
  MoveL 9652 to (238.75, 43.06, 135.08) mm, rotated rx -180 ry 0 rz 180 deg; joints [-28.669, 57.845, -90.493, 32.998, 118.251, 17.086]
  Call Extruder(199.83852)
  MoveL 9653 to (238.89, 43.34, 135.08) mm, rotated rx 180 ry 0 rz 180 deg; joints [-28.78, 57.875, -90.491, 33.11, 118.192, 17.124]
  MoveL 9654 to (238.89, 43.34, 135.08) mm, rotated rx 180 ry 0 rz 180 deg; joints [-28.78, 57.875, -90.491, 33.11, 118.192, 17.124]
  Call Extruder(199.99654)
  MoveL 9655 to (239, 43.58, 135.08) mm, rotated rx -180 ry 0 rz 180 deg; joints [-28.886, 57.899, -90.49, 33.217, 118.139, 17.162]
  MoveL 9656 to (239, 43.58, 135.08) mm, rotated rx -180 ry 0 rz 180 deg; joints [-28.886, 57.899, -90.49, 33.217, 118.139, 17.162]
  Call Extruder(200.15395)
  MoveL 9657 to (239.11, 43.83, 135.08) mm, rotated rx 180 ry 0 rz -180 deg; joints [-28.991, 57.924, -90.488, 33.324, 118.087, 17.2]
  MoveL 9658 to (239.11, 43.83, 135.08) mm, rotated rx 180 ry 0 rz -180 deg; joints [-28.991, 57.924, -90.488, 33.324, 118.087, 17.2]
  Call Extruder(200.33666)
  MoveL 9659 to (239.22, 44.12, 135.08) mm, rotated rx -180 ry 0 rz 180 deg; joints [-29.116, 57.952, -90.487, 33.45, 118.025, 17.245]
  MoveL 9660 to (239.22, 44.12, 135.08) mm, rotated rx -180 ry 0 rz 180 deg; joints [-29.116, 57.952, -90.487, 33.45, 118.025, 17.245]
  Call Extruder(200.51862)
  MoveL 9661 to (239.35, 44.42, 135.08) mm, rotated rx -180 ry 0 rz -180 deg; joints [-29.24, 57.98, -90.485, 33.575, 117.963, 17.289]
  MoveL 9662 to (239.35, 44.42, 135.08) mm, rotated rx -180 ry 0 rz -180 deg; joints [-29.24, 57.98, -90.485, 33.575, 117.963, 17.289]
  Call Extruder(200.66595)
  MoveL 9663 to (239.44, 44.66, 135.08) mm, rotated rx 180 ry 0 rz -180 deg; joints [-29.343, 58.003, -90.484, 33.68, 117.913, 17.326]
  MoveL 9664 to (239.44, 44.66, 135.08) mm, rotated rx 180 ry 0 rz -180 deg; joints [-29.343, 58.003, -90.484, 33.68, 117.913, 17.326]
  Call Extruder(200.77919)
  MoveL 9665 to (239.5, 44.85, 135.08) mm, rotated rx -180 ry 0 rz 180 deg; joints [-29.428, 58.019, -90.483, 33.766, 117.873, 17.358]
  MoveL 9666 to (239.5, 44.85, 135.08) mm, rotated rx -180 ry 0 rz 180 deg; joints [-29.428, 58.019, -90.483, 33.766, 117.873, 17.358]
  Call Extruder(200.89198)
  MoveL 9667 to (239.56, 45.03, 135.08) mm, rotated rx -180 ry 0 rz -180 deg; joints [-29.512, 58.036, -90.482, 33.852, 117.833, 17.389]
  MoveL 9668 to (239.56, 45.03, 135.08) mm, rotated rx -180 ry 0 rz -180 deg; joints [-29.512, 58.036, -90.482, 33.852, 117.833, 17.389]
  Call Extruder(201.00432)
  MoveL 9669 to (239.62, 45.22, 135.08) mm, rotated rx -180 ry 0 rz 180 deg; joints [-29.596, 58.053, -90.481, 33.937, 117.794, 17.42]
  MoveL 9670 to (239.62, 45.22, 135.08) mm, rotated rx -180 ry 0 rz 180 deg; joints [-29.596, 58.053, -90.481, 33.937, 117.794, 17.42]
  Call Extruder(201.11622)
  MoveL 9671 to (239.68, 45.41, 135.08) mm, rotated rx 180 ry 0 rz 180 deg; joints [-29.679, 58.069, -90.481, 34.022, 117.754, 17.451]
  MoveL 9672 to (239.68, 45.41, 135.08) mm, rotated rx 180 ry 0 rz 180 deg; joints [-29.679, 58.069, -90.481, 34.022, 117.754, 17.451]
  Call Extruder(201.23762)
  MoveL 9673 to (239.75, 45.62, 135.08) mm, rotated rx 180 ry 0 rz 180 deg; joints [-29.77, 58.087, -90.479, 34.115, 117.711, 17.485]
  MoveL 9674 to (239.75, 45.62, 135.08) mm, rotated rx 180 ry 0 rz 180 deg; joints [-29.77, 58.087, -90.479, 34.115, 117.711, 17.485]
  Call Extruder(201.36842)
  MoveL 9675 to (239.82, 45.84, 135.08) mm, rotated rx 180 ry 0 rz 180 deg; joints [-29.871, 58.107, -90.478, 34.217, 117.664, 17.522]
  MoveL 9676 to (239.82, 45.84, 135.08) mm, rotated rx 180 ry 0 rz 180 deg; joints [-29.871, 58.107, -90.478, 34.217, 117.664, 17.522]
  Call Extruder(201.49864)
  MoveL 9677 to (239.88, 46.06, 135.08) mm, rotated rx 180 ry 0 rz 180 deg; joints [-29.97, 58.126, -90.477, 34.318, 117.617, 17.559]
  MoveL 9678 to (239.88, 46.06, 135.08) mm, rotated rx 180 ry 0 rz 180 deg; joints [-29.97, 58.126, -90.477, 34.318, 117.617, 17.559]
  Call Extruder(201.62830)
  MoveL 9679 to (239.95, 46.29, 135.08) mm, rotated rx -180 ry 0 rz -180 deg; joints [-30.069, 58.145, -90.476, 34.418, 117.57, 17.595]
  MoveL 9680 to (239.95, 46.29, 135.08) mm, rotated rx -180 ry 0 rz -180 deg; joints [-30.069, 58.145, -90.476, 34.418, 117.57, 17.595]
  Call Extruder(201.75740)
  MoveL 9681 to (240.02, 46.51, 135.08) mm, rotated rx -180 ry 0 rz 180 deg; joints [-30.168, 58.165, -90.475, 34.519, 117.523, 17.631]
  MoveL 9682 to (240.02, 46.51, 135.08) mm, rotated rx -180 ry 0 rz 180 deg; joints [-30.168, 58.165, -90.475, 34.519, 117.523, 17.631]
  Call Extruder(201.87246)
  MoveL 9683 to (240.06, 46.72, 135.08) mm, rotated rx -180 ry 0 rz 180 deg; joints [-30.263, 58.181, -90.474, 34.616, 117.48, 17.668]
  MoveL 9684 to (240.06, 46.72, 135.08) mm, rotated rx -180 ry 0 rz 180 deg; joints [-30.263, 58.181, -90.474, 34.616, 117.48, 17.668]
  Call Extruder(201.98706)
  MoveL 9685 to (240.11, 46.92, 135.08) mm, rotated rx -180 ry 0 rz 180 deg; joints [-30.358, 58.197, -90.473, 34.713, 117.437, 17.704]
  MoveL 9686 to (240.11, 46.92, 135.08) mm, rotated rx -180 ry 0 rz 180 deg; joints [-30.358, 58.197, -90.473, 34.713, 117.437, 17.704]
  Call Extruder(202.10121)
  MoveL 9687 to (240.15, 47.12, 135.08) mm, rotated rx 180 ry 0 rz 180 deg; joints [-30.453, 58.213, -90.472, 34.809, 117.395, 17.739]
  MoveL 9688 to (240.15, 47.12, 135.08) mm, rotated rx 180 ry 0 rz 180 deg; joints [-30.453, 58.213, -90.472, 34.809, 117.395, 17.739]
  Call Extruder(202.21491)
  MoveL 9689 to (240.2, 47.33, 135.08) mm, rotated rx 180 ry 0 rz 180 deg; joints [-30.548, 58.229, -90.471, 34.906, 117.352, 17.775]
  MoveL 9690 to (240.2, 47.33, 135.08) mm, rotated rx 180 ry 0 rz 180 deg; joints [-30.548, 58.229, -90.471, 34.906, 117.352, 17.775]
  Call Extruder(202.34032)
  MoveL 9691 to (240.24, 47.55, 135.08) mm, rotated rx 180 ry 0 rz 180 deg; joints [-30.653, 58.247, -90.47, 35.013, 117.304, 17.815]
  MoveL 9692 to (240.24, 47.55, 135.08) mm, rotated rx 180 ry 0 rz 180 deg; joints [-30.653, 58.247, -90.47, 35.013, 117.304, 17.815]
  Call Extruder(202.47730)
  MoveL 9693 to (240.29, 47.8, 135.08) mm, rotated rx -180 ry 0 rz 180 deg; joints [-30.768, 58.266, -90.469, 35.13, 117.252, 17.858]
  MoveL 9694 to (240.29, 47.8, 135.08) mm, rotated rx -180 ry 0 rz 180 deg; joints [-30.768, 58.266, -90.469, 35.13, 117.252, 17.858]
  Call Extruder(202.61366)
  MoveL 9695 to (240.34, 48.05, 135.08) mm, rotated rx -180 ry 0 rz 180 deg; joints [-30.884, 58.285, -90.467, 35.248, 117.2, 17.901]
  MoveL 9696 to (240.34, 48.05, 135.08) mm, rotated rx -180 ry 0 rz 180 deg; joints [-30.884, 58.285, -90.467, 35.248, 117.2, 17.901]
  Call Extruder(202.74942)
  MoveL 9697 to (240.39, 48.3, 135.08) mm, rotated rx 180 ry 0 rz 180 deg; joints [-30.999, 58.305, -90.466, 35.365, 117.147, 17.944]
  MoveL 9698 to (240.39, 48.3, 135.08) mm, rotated rx 180 ry 0 rz 180 deg; joints [-30.999, 58.305, -90.466, 35.365, 117.147, 17.944]
  Call Extruder(202.88457)
  MoveL 9699 to (240.44, 48.55, 135.08) mm, rotated rx 180 ry 0 rz 180 deg; joints [-31.114, 58.324, -90.465, 35.482, 117.095, 17.987]
  MoveL 9700 to (240.44, 48.55, 135.08) mm, rotated rx 180 ry 0 rz 180 deg; joints [-31.114, 58.324, -90.465, 35.482, 117.095, 17.987]
  Call Extruder(203.01910)
  MoveL 9701 to (240.49, 48.8, 135.08) mm, rotated rx -180 ry 0 rz 180 deg; joints [-31.228, 58.343, -90.464, 35.598, 117.043, 18.029]
  MoveL 9702 to (240.49, 48.8, 135.08) mm, rotated rx -180 ry 0 rz 180 deg; joints [-31.228, 58.343, -90.464, 35.598, 117.043, 18.029]
  Call Extruder(203.15303)
  MoveL 9703 to (240.54, 49.05, 135.08) mm, rotated rx -180 ry 0 rz 180 deg; joints [-31.342, 58.363, -90.462, 35.713, 116.991, 18.071]
  MoveL 9704 to (240.54, 49.05, 135.08) mm, rotated rx -180 ry 0 rz 180 deg; joints [-31.342, 58.363, -90.462, 35.713, 116.991, 18.071]
  Call Extruder(203.30090)
  MoveL 9705 to (240.59, 49.33, 135.08) mm, rotated rx 180 ry 0 rz 180 deg; joints [-31.47, 58.384, -90.461, 35.843, 116.933, 18.118]
  MoveL 9706 to (240.59, 49.33, 135.08) mm, rotated rx 180 ry 0 rz 180 deg; joints [-31.47, 58.384, -90.461, 35.843, 116.933, 18.118]
  Call Extruder(203.46264)
  MoveL 9707 to (240.64, 49.63, 135.08) mm, rotated rx 180 ry 0 rz 180 deg; joints [-31.612, 58.407, -90.46, 35.987, 116.869, 18.17]
  MoveL 9708 to (240.64, 49.63, 135.08) mm, rotated rx 180 ry 0 rz 180 deg; joints [-31.612, 58.407, -90.46, 35.987, 116.869, 18.17]
  Call Extruder(203.62365)
  MoveL 9709 to (240.69, 49.94, 135.08) mm, rotated rx -180 ry 0 rz 180 deg; joints [-31.755, 58.429, -90.458, 36.132, 116.805, 18.223]
  MoveL 9710 to (240.69, 49.94, 135.08) mm, rotated rx -180 ry 0 rz 180 deg; joints [-31.755, 58.429, -90.458, 36.132, 116.805, 18.223]
  Call Extruder(203.78394)
  MoveL 9711 to (240.74, 50.24, 135.08) mm, rotated rx -180 ry 0 rz 180 deg; joints [-31.895, 58.452, -90.456, 36.274, 116.741, 18.274]
  MoveL 9712 to (240.74, 50.24, 135.08) mm, rotated rx -180 ry 0 rz 180 deg; joints [-31.895, 58.452, -90.456, 36.274, 116.741, 18.274]
  Call Extruder(203.94350)
  MoveL 9713 to (240.78, 50.55, 135.08) mm, rotated rx -180 ry 0 rz 180 deg; joints [-32.036, 58.475, -90.455, 36.416, 116.677, 18.325]
  MoveL 9714 to (240.78, 50.55, 135.08) mm, rotated rx -180 ry 0 rz 180 deg; joints [-32.036, 58.475, -90.455, 36.416, 116.677, 18.325]
  Call Extruder(204.10233)
  MoveL 9715 to (240.83, 50.86, 135.08) mm, rotated rx -180 ry 0 rz 180 deg; joints [-32.176, 58.498, -90.453, 36.558, 116.613, 18.375]
  MoveL 9716 to (240.83, 50.86, 135.08) mm, rotated rx -180 ry 0 rz 180 deg; joints [-32.176, 58.498, -90.453, 36.558, 116.613, 18.375]
  Call Extruder(204.28100)
  MoveL 9717 to (240.88, 51.2, 135.08) mm, rotated rx 180 ry 0 rz 180 deg; joints [-32.337, 58.524, -90.451, 36.72, 116.541, 18.433]
  MoveL 9718 to (240.88, 51.2, 135.08) mm, rotated rx 180 ry 0 rz 180 deg; joints [-32.337, 58.524, -90.451, 36.72, 116.541, 18.433]
  Call Extruder(204.47945)
  MoveL 9719 to (240.93, 51.59, 135.08) mm, rotated rx 180 ry 0 rz 180 deg; joints [-32.518, 58.551, -90.449, 36.903, 116.46, 18.499]
  MoveL 9720 to (240.93, 51.59, 135.08) mm, rotated rx 180 ry 0 rz 180 deg; joints [-32.518, 58.551, -90.449, 36.903, 116.46, 18.499]
  Call Extruder(204.67702)
  MoveL 9721 to (240.97, 51.98, 135.08) mm, rotated rx -180 ry 0 rz 180 deg; joints [-32.697, 58.579, -90.447, 37.084, 116.379, 18.563]
  MoveL 9722 to (240.97, 51.98, 135.08) mm, rotated rx -180 ry 0 rz 180 deg; joints [-32.697, 58.579, -90.447, 37.084, 116.379, 18.563]
  Call Extruder(204.87373)
  MoveL 9723 to (241.02, 52.37, 135.08) mm, rotated rx -180 ry 0 rz -180 deg; joints [-32.876, 58.607, -90.445, 37.264, 116.298, 18.627]
  MoveL 9724 to (241.02, 52.37, 135.08) mm, rotated rx -180 ry 0 rz -180 deg; joints [-32.876, 58.607, -90.445, 37.264, 116.298, 18.627]
  Call Extruder(205.06957)
  MoveL 9725 to (241.06, 52.75, 135.08) mm, rotated rx 180 ry 0 rz 180 deg; joints [-33.055, 58.635, -90.443, 37.444, 116.217, 18.69]
  MoveL 9726 to (241.06, 52.75, 135.08) mm, rotated rx 180 ry 0 rz 180 deg; joints [-33.055, 58.635, -90.443, 37.444, 116.217, 18.69]
  Call Extruder(205.36500)
  MoveL 9727 to (241.11, 53.34, 135.08) mm, rotated rx 180 ry 0 rz -180 deg; joints [-33.331, 58.676, -90.44, 37.722, 116.093, 18.789]
  MoveL 9728 to (241.11, 53.34, 135.08) mm, rotated rx 180 ry 0 rz -180 deg; joints [-33.331, 58.676, -90.44, 37.722, 116.093, 18.789]
  Call Extruder(205.65911)
  MoveL 9729 to (241.15, 53.93, 135.08) mm, rotated rx -180 ry 0 rz 180 deg; joints [-33.606, 58.717, -90.437, 37.998, 115.97, 18.886]
  MoveL 9730 to (241.15, 53.93, 135.08) mm, rotated rx -180 ry 0 rz 180 deg; joints [-33.606, 58.717, -90.437, 37.998, 115.97, 18.886]
  Call Extruder(205.95189)
  MoveL 9731 to (241.2, 54.52, 135.08) mm, rotated rx 180 ry 0 rz 180 deg; joints [-33.878, 58.758, -90.434, 38.272, 115.846, 18.981]
  MoveL 9732 to (241.2, 54.52, 135.08) mm, rotated rx 180 ry 0 rz 180 deg; joints [-33.878, 58.758, -90.434, 38.272, 115.846, 18.981]
  Call Extruder(206.52534)
  MoveL 9733 to (241.25, 55.68, 135.08) mm, rotated rx 180 ry 0 rz 180 deg; joints [-34.425, 58.836, -90.428, 38.82, 115.602, 19.171]
  MoveL 9734 to (241.25, 55.68, 135.08) mm, rotated rx 180 ry 0 rz 180 deg; joints [-34.425, 58.836, -90.428, 38.82, 115.602, 19.171]
  Call Extruder(207.23917)
  MoveL 9735 to (241.29, 57.14, 135.08) mm, rotated rx 180 ry 0 rz 180 deg; joints [-35.104, 58.932, -90.42, 39.498, 115.297, 19.404]
  Call Extruder(249.30405)
  MoveL 9736 to (241.29, 142.86, 135.08) mm, rotated rx -180 ry 0 rz 180 deg; joints [-60.361, 65.64, -88.988, 62.418, 101.303, 20.565]
  Call Extruder(249.73248)
  MoveL 9737 to (241.27, 143.74, 135.08) mm, rotated rx 180 ry 0 rz 180 deg; joints [-60.516, 65.711, -88.962, 62.548, 101.204, 20.507]
  MoveL 9738 to (241.27, 143.74, 135.08) mm, rotated rx 180 ry 0 rz 180 deg; joints [-60.516, 65.711, -88.962, 62.548, 101.204, 20.507]
  Call Extruder(250.30594)
  MoveL 9739 to (241.22, 144.9, 135.08) mm, rotated rx -180 ry 0 rz 180 deg; joints [-60.726, 65.804, -88.928, 62.728, 101.071, 20.43]
  MoveL 9740 to (241.22, 144.9, 135.08) mm, rotated rx -180 ry 0 rz 180 deg; joints [-60.726, 65.804, -88.928, 62.728, 101.071, 20.43]
  Call Extruder(250.74027)
  MoveL 9741 to (241.18, 145.77, 135.08) mm, rotated rx 180 ry 0 rz 180 deg; joints [-60.887, 65.873, -88.901, 62.865, 100.972, 20.373]
  MoveL 9742 to (241.18, 145.77, 135.08) mm, rotated rx 180 ry 0 rz 180 deg; joints [-60.887, 65.873, -88.901, 62.865, 100.972, 20.373]
  Call Extruder(251.03438)
  MoveL 9743 to (241.13, 146.36, 135.08) mm, rotated rx 180 ry 0 rz -180 deg; joints [-61, 65.919, -88.884, 62.961, 100.904, 20.336]
  MoveL 9744 to (241.13, 146.36, 135.08) mm, rotated rx 180 ry 0 rz -180 deg; joints [-61, 65.919, -88.884, 62.961, 100.904, 20.336]
  Call Extruder(251.32982)
  MoveL 9745 to (241.09, 146.95, 135.08) mm, rotated rx -180 ry 0 rz 180 deg; joints [-61.111, 65.964, -88.866, 63.056, 100.836, 20.299]
  MoveL 9746 to (241.09, 146.95, 135.08) mm, rotated rx -180 ry 0 rz 180 deg; joints [-61.111, 65.964, -88.866, 63.056, 100.836, 20.299]
  Call Extruder(251.57607)
  MoveL 9747 to (241.04, 147.44, 135.08) mm, rotated rx -180 ry 0 rz 180 deg; joints [-61.205, 66.002, -88.852, 63.137, 100.78, 20.268]
  MoveL 9748 to (241.04, 147.44, 135.08) mm, rotated rx -180 ry 0 rz 180 deg; joints [-61.205, 66.002, -88.852, 63.137, 100.78, 20.268]
  Call Extruder(251.77278)
  MoveL 9749 to (240.99, 147.83, 135.08) mm, rotated rx -180 ry 0 rz -180 deg; joints [-61.282, 66.032, -88.84, 63.204, 100.735, 20.245]
  MoveL 9750 to (240.99, 147.83, 135.08) mm, rotated rx -180 ry 0 rz -180 deg; joints [-61.282, 66.032, -88.84, 63.204, 100.735, 20.245]
  Call Extruder(251.97035)
  MoveL 9751 to (240.95, 148.22, 135.08) mm, rotated rx -180 ry 0 rz 180 deg; joints [-61.359, 66.061, -88.829, 63.27, 100.69, 20.221]
  MoveL 9752 to (240.95, 148.22, 135.08) mm, rotated rx -180 ry 0 rz 180 deg; joints [-61.359, 66.061, -88.829, 63.27, 100.69, 20.221]
  Call Extruder(252.16879)
  MoveL 9753 to (240.9, 148.6, 135.08) mm, rotated rx -180 ry 0 rz 180 deg; joints [-61.436, 66.09, -88.817, 63.337, 100.645, 20.197]
  MoveL 9754 to (240.9, 148.6, 135.08) mm, rotated rx -180 ry 0 rz 180 deg; joints [-61.436, 66.09, -88.817, 63.337, 100.645, 20.197]
  Call Extruder(252.36810)
  MoveL 9755 to (240.86, 148.99, 135.08) mm, rotated rx -180 ry 0 rz 180 deg; joints [-61.512, 66.12, -88.806, 63.403, 100.601, 20.173]
  MoveL 9756 to (240.86, 148.99, 135.08) mm, rotated rx -180 ry 0 rz 180 deg; joints [-61.512, 66.12, -88.806, 63.403, 100.601, 20.173]
  Call Extruder(252.52693)
  MoveL 9757 to (240.81, 149.3, 135.08) mm, rotated rx 180 ry 0 rz 180 deg; joints [-61.575, 66.142, -88.797, 63.458, 100.564, 20.156]
  MoveL 9758 to (240.81, 149.3, 135.08) mm, rotated rx 180 ry 0 rz 180 deg; joints [-61.575, 66.142, -88.797, 63.458, 100.564, 20.156]
  Call Extruder(252.68649)
  MoveL 9759 to (240.76, 149.6, 135.08) mm, rotated rx -180 ry 0 rz 180 deg; joints [-61.639, 66.165, -88.788, 63.513, 100.528, 20.138]
  MoveL 9760 to (240.76, 149.6, 135.08) mm, rotated rx -180 ry 0 rz 180 deg; joints [-61.639, 66.165, -88.788, 63.513, 100.528, 20.138]
  Call Extruder(252.84678)
  MoveL 9761 to (240.71, 149.91, 135.08) mm, rotated rx 180 ry 0 rz 180 deg; joints [-61.702, 66.188, -88.779, 63.568, 100.493, 20.12]
  MoveL 9762 to (240.71, 149.91, 135.08) mm, rotated rx 180 ry 0 rz 180 deg; joints [-61.702, 66.188, -88.779, 63.568, 100.493, 20.12]
  Call Extruder(253.00780)
  MoveL 9763 to (240.66, 150.21, 135.08) mm, rotated rx -180 ry 0 rz 180 deg; joints [-61.765, 66.21, -88.77, 63.623, 100.457, 20.102]
  MoveL 9764 to (240.66, 150.21, 135.08) mm, rotated rx -180 ry 0 rz 180 deg; joints [-61.765, 66.21, -88.77, 63.623, 100.457, 20.102]
  Call Extruder(253.16954)
  MoveL 9765 to (240.61, 150.52, 135.08) mm, rotated rx -180 ry 0 rz 180 deg; joints [-61.828, 66.233, -88.76, 63.678, 100.421, 20.084]
  MoveL 9766 to (240.61, 150.52, 135.08) mm, rotated rx -180 ry 0 rz 180 deg; joints [-61.828, 66.233, -88.76, 63.678, 100.421, 20.084]
  Call Extruder(253.33202)
  MoveL 9767 to (240.56, 150.83, 135.08) mm, rotated rx -180 ry 0 rz 180 deg; joints [-61.891, 66.256, -88.751, 63.733, 100.385, 20.066]
  MoveL 9768 to (240.56, 150.83, 135.08) mm, rotated rx -180 ry 0 rz 180 deg; joints [-61.891, 66.256, -88.751, 63.733, 100.385, 20.066]
  Call Extruder(253.46594)
  MoveL 9769 to (240.52, 151.08, 135.08) mm, rotated rx 180 ry 0 rz -180 deg; joints [-61.944, 66.274, -88.744, 63.78, 100.356, 20.052]
  MoveL 9770 to (240.52, 151.08, 135.08) mm, rotated rx 180 ry 0 rz -180 deg; joints [-61.944, 66.274, -88.744, 63.78, 100.356, 20.052]
  Call Extruder(253.60048)
  MoveL 9771 to (240.47, 151.32, 135.08) mm, rotated rx 180 ry 0 rz -180 deg; joints [-61.998, 66.292, -88.737, 63.827, 100.326, 20.038]
  MoveL 9772 to (240.47, 151.32, 135.08) mm, rotated rx 180 ry 0 rz -180 deg; joints [-61.998, 66.292, -88.737, 63.827, 100.326, 20.038]
  Call Extruder(253.73563)
  MoveL 9773 to (240.42, 151.57, 135.08) mm, rotated rx 180 ry 0 rz 180 deg; joints [-62.052, 66.31, -88.729, 63.875, 100.297, 20.024]
  MoveL 9774 to (240.42, 151.57, 135.08) mm, rotated rx 180 ry 0 rz 180 deg; joints [-62.052, 66.31, -88.729, 63.875, 100.297, 20.024]
  Call Extruder(253.87138)
  MoveL 9775 to (240.37, 151.82, 135.08) mm, rotated rx 180 ry 0 rz -180 deg; joints [-62.105, 66.328, -88.722, 63.922, 100.267, 20.01]
  MoveL 9776 to (240.37, 151.82, 135.08) mm, rotated rx 180 ry 0 rz -180 deg; joints [-62.105, 66.328, -88.722, 63.922, 100.267, 20.01]
  Call Extruder(254.00775)
  MoveL 9777 to (240.32, 152.07, 135.08) mm, rotated rx -180 ry 0 rz 180 deg; joints [-62.159, 66.346, -88.715, 63.969, 100.238, 19.996]
  MoveL 9778 to (240.32, 152.07, 135.08) mm, rotated rx -180 ry 0 rz 180 deg; joints [-62.159, 66.346, -88.715, 63.969, 100.238, 19.996]
  Call Extruder(254.14473)
  MoveL 9779 to (240.27, 152.32, 135.08) mm, rotated rx 180 ry 0 rz 180 deg; joints [-62.212, 66.364, -88.707, 64.015, 100.208, 19.982]
  MoveL 9780 to (240.27, 152.32, 135.08) mm, rotated rx 180 ry 0 rz 180 deg; joints [-62.212, 66.364, -88.707, 64.015, 100.208, 19.982]
  Call Extruder(254.28232)
  MoveL 9781 to (240.22, 152.57, 135.08) mm, rotated rx -180 ry 0 rz 180 deg; joints [-62.265, 66.382, -88.7, 64.062, 100.179, 19.968]
  MoveL 9782 to (240.22, 152.57, 135.08) mm, rotated rx -180 ry 0 rz 180 deg; joints [-62.265, 66.382, -88.7, 64.062, 100.179, 19.968]
  Call Extruder(254.39601)
  MoveL 9783 to (240.17, 152.77, 135.08) mm, rotated rx -180 ry 0 rz 180 deg; joints [-62.31, 66.397, -88.694, 64.101, 100.155, 19.956]
  MoveL 9784 to (240.17, 152.77, 135.08) mm, rotated rx -180 ry 0 rz 180 deg; joints [-62.31, 66.397, -88.694, 64.101, 100.155, 19.956]
  Call Extruder(254.51016)
  MoveL 9785 to (240.13, 152.98, 135.08) mm, rotated rx -180 ry 0 rz 180 deg; joints [-62.355, 66.411, -88.688, 64.14, 100.13, 19.945]
  MoveL 9786 to (240.13, 152.98, 135.08) mm, rotated rx -180 ry 0 rz 180 deg; joints [-62.355, 66.411, -88.688, 64.14, 100.13, 19.945]
  Call Extruder(254.62477)
  MoveL 9787 to (240.08, 153.18, 135.08) mm, rotated rx -180 ry 0 rz 180 deg; joints [-62.399, 66.426, -88.682, 64.18, 100.106, 19.934]
  MoveL 9788 to (240.08, 153.18, 135.08) mm, rotated rx -180 ry 0 rz 180 deg; joints [-62.399, 66.426, -88.682, 64.18, 100.106, 19.934]
  Call Extruder(254.73982)
  MoveL 9789 to (240.04, 153.39, 135.08) mm, rotated rx -180 ry 0 rz -180 deg; joints [-62.444, 66.441, -88.676, 64.219, 100.082, 19.922]
  MoveL 9790 to (240.04, 153.39, 135.08) mm, rotated rx -180 ry 0 rz -180 deg; joints [-62.444, 66.441, -88.676, 64.219, 100.082, 19.922]
  Call Extruder(254.86204)
  MoveL 9791 to (239.98, 153.6, 135.08) mm, rotated rx -180 ry 0 rz 180 deg; joints [-62.493, 66.456, -88.67, 64.262, 100.056, 19.911]
  MoveL 9792 to (239.98, 153.6, 135.08) mm, rotated rx -180 ry 0 rz 180 deg; joints [-62.493, 66.456, -88.67, 64.262, 100.056, 19.911]
  Call Extruder(254.99170)
  MoveL 9793 to (239.92, 153.82, 135.08) mm, rotated rx -180 ry 0 rz 180 deg; joints [-62.547, 66.471, -88.663, 64.31, 100.028, 19.9]
  MoveL 9794 to (239.92, 153.82, 135.08) mm, rotated rx -180 ry 0 rz 180 deg; joints [-62.547, 66.471, -88.663, 64.31, 100.028, 19.9]
  Call Extruder(255.12193)
  MoveL 9795 to (239.85, 154.05, 135.08) mm, rotated rx -180 ry 0 rz 180 deg; joints [-62.601, 66.486, -88.657, 64.358, 100.001, 19.889]
  MoveL 9796 to (239.85, 154.05, 135.08) mm, rotated rx -180 ry 0 rz 180 deg; joints [-62.601, 66.486, -88.657, 64.358, 100.001, 19.889]
  Call Extruder(255.25272)
  MoveL 9797 to (239.78, 154.27, 135.08) mm, rotated rx 180 ry 0 rz -180 deg; joints [-62.654, 66.501, -88.651, 64.406, 99.973, 19.878]
  MoveL 9798 to (239.78, 154.27, 135.08) mm, rotated rx 180 ry 0 rz -180 deg; joints [-62.654, 66.501, -88.651, 64.406, 99.973, 19.878]
  Call Extruder(255.38407)
  MoveL 9799 to (239.71, 154.49, 135.08) mm, rotated rx -180 ry 0 rz 180 deg; joints [-62.708, 66.517, -88.644, 64.454, 99.945, 19.867]
  MoveL 9800 to (239.71, 154.49, 135.08) mm, rotated rx -180 ry 0 rz 180 deg; joints [-62.708, 66.517, -88.644, 64.454, 99.945, 19.867]
  Call Extruder(255.49598)
  MoveL 9801 to (239.65, 154.68, 135.08) mm, rotated rx -180 ry 0 rz 180 deg; joints [-62.754, 66.529, -88.639, 64.496, 99.922, 19.859]
  MoveL 9802 to (239.65, 154.68, 135.08) mm, rotated rx -180 ry 0 rz 180 deg; joints [-62.754, 66.529, -88.639, 64.496, 99.922, 19.859]
  Call Extruder(255.60832)
  MoveL 9803 to (239.59, 154.87, 135.08) mm, rotated rx -180 ry 0 rz 180 deg; joints [-62.801, 66.542, -88.633, 64.537, 99.899, 19.85]
  MoveL 9804 to (239.59, 154.87, 135.08) mm, rotated rx -180 ry 0 rz 180 deg; joints [-62.801, 66.542, -88.633, 64.537, 99.899, 19.85]
  Call Extruder(255.72111)
  MoveL 9805 to (239.53, 155.06, 135.08) mm, rotated rx -180 ry 0 rz 180 deg; joints [-62.847, 66.555, -88.628, 64.578, 99.875, 19.841]
  MoveL 9806 to (239.53, 155.06, 135.08) mm, rotated rx -180 ry 0 rz 180 deg; joints [-62.847, 66.555, -88.628, 64.578, 99.875, 19.841]
  Call Extruder(255.83435)
  MoveL 9807 to (239.47, 155.25, 135.08) mm, rotated rx -180 ry 0 rz 180 deg; joints [-62.893, 66.567, -88.623, 64.62, 99.852, 19.832]
  MoveL 9808 to (239.47, 155.25, 135.08) mm, rotated rx -180 ry 0 rz 180 deg; joints [-62.893, 66.567, -88.623, 64.62, 99.852, 19.832]
  Call Extruder(255.94803)
  MoveL 9809 to (239.41, 155.44, 135.08) mm, rotated rx -180 ry 0 rz -180 deg; joints [-62.939, 66.58, -88.617, 64.661, 99.828, 19.823]
  MoveL 9810 to (239.41, 155.44, 135.08) mm, rotated rx -180 ry 0 rz -180 deg; joints [-62.939, 66.58, -88.617, 64.661, 99.828, 19.823]
  Call Extruder(256.12998)
  MoveL 9811 to (239.29, 155.73, 135.08) mm, rotated rx -180 ry 0 rz 180 deg; joints [-63.018, 66.599, -88.61, 64.732, 99.79, 19.811]
  MoveL 9812 to (239.29, 155.73, 135.08) mm, rotated rx -180 ry 0 rz 180 deg; joints [-63.018, 66.599, -88.61, 64.732, 99.79, 19.811]
  Call Extruder(256.31270)
  MoveL 9813 to (239.16, 156.02, 135.08) mm, rotated rx -180 ry 0 rz 180 deg; joints [-63.097, 66.617, -88.602, 64.803, 99.752, 19.8]
  MoveL 9814 to (239.16, 156.02, 135.08) mm, rotated rx -180 ry 0 rz 180 deg; joints [-63.097, 66.617, -88.602, 64.803, 99.752, 19.8]
  Call Extruder(256.48312)
  MoveL 9815 to (239.05, 156.29, 135.08) mm, rotated rx 180 ry 0 rz 180 deg; joints [-63.17, 66.635, -88.594, 64.869, 99.717, 19.789]
  MoveL 9816 to (239.05, 156.29, 135.08) mm, rotated rx 180 ry 0 rz 180 deg; joints [-63.17, 66.635, -88.594, 64.869, 99.717, 19.789]
  Call Extruder(256.64113)
  MoveL 9817 to (238.94, 156.54, 135.08) mm, rotated rx -180 ry 0 rz -180 deg; joints [-63.238, 66.65, -88.588, 64.93, 99.685, 19.779]
  MoveL 9818 to (238.94, 156.54, 135.08) mm, rotated rx -180 ry 0 rz -180 deg; joints [-63.238, 66.65, -88.588, 64.93, 99.685, 19.779]
  Call Extruder(256.79975)
  MoveL 9819 to (238.84, 156.79, 135.08) mm, rotated rx -180 ry 0 rz -180 deg; joints [-63.306, 66.666, -88.581, 64.992, 99.652, 19.769]
  MoveL 9820 to (238.84, 156.79, 135.08) mm, rotated rx -180 ry 0 rz -180 deg; joints [-63.306, 66.666, -88.581, 64.992, 99.652, 19.769]
  Call Extruder(257.00592)
  MoveL 9821 to (238.66, 157.09, 135.08) mm, rotated rx 180 ry 0 rz 180 deg; joints [-63.401, 66.684, -88.573, 65.079, 99.609, 19.762]
  MoveL 9822 to (238.66, 157.09, 135.08) mm, rotated rx 180 ry 0 rz 180 deg; joints [-63.401, 66.684, -88.573, 65.079, 99.609, 19.762]
  Call Extruder(257.21287)
  MoveL 9823 to (238.49, 157.4, 135.08) mm, rotated rx 180 ry 0 rz 180 deg; joints [-63.497, 66.701, -88.566, 65.166, 99.566, 19.754]
  MoveL 9824 to (238.49, 157.4, 135.08) mm, rotated rx 180 ry 0 rz 180 deg; joints [-63.497, 66.701, -88.566, 65.166, 99.566, 19.754]
  Call Extruder(257.42059)
  MoveL 9825 to (238.31, 157.7, 135.08) mm, rotated rx 180 ry 0 rz 180 deg; joints [-63.592, 66.719, -88.558, 65.253, 99.524, 19.746]
  MoveL 9826 to (238.31, 157.7, 135.08) mm, rotated rx 180 ry 0 rz 180 deg; joints [-63.592, 66.719, -88.558, 65.253, 99.524, 19.746]
  Call Extruder(257.62910)
  MoveL 9827 to (238.14, 158.01, 135.08) mm, rotated rx -180 ry 0 rz -180 deg; joints [-63.687, 66.736, -88.551, 65.34, 99.481, 19.738]
  MoveL 9828 to (238.14, 158.01, 135.08) mm, rotated rx -180 ry 0 rz -180 deg; joints [-63.687, 66.736, -88.551, 65.34, 99.481, 19.738]
  Call Extruder(257.80864)
  MoveL 9829 to (237.96, 158.25, 135.08) mm, rotated rx -180 ry 0 rz 180 deg; joints [-63.774, 66.749, -88.545, 65.42, 99.444, 19.734]
  MoveL 9830 to (237.96, 158.25, 135.08) mm, rotated rx -180 ry 0 rz 180 deg; joints [-63.774, 66.749, -88.545, 65.42, 99.444, 19.734]
  Call Extruder(258.14205)
  MoveL 9831 to (237.63, 158.7, 135.08) mm, rotated rx -180 ry 0 rz -180 deg; joints [-63.934, 66.772, -88.535, 65.568, 99.376, 19.728]
  MoveL 9832 to (237.63, 158.7, 135.08) mm, rotated rx -180 ry 0 rz -180 deg; joints [-63.934, 66.772, -88.535, 65.568, 99.376, 19.728]
  Call Extruder(258.47664)
  MoveL 9833 to (237.3, 159.15, 135.08) mm, rotated rx 180 ry 0 rz 180 deg; joints [-64.094, 66.796, -88.525, 65.715, 99.308, 19.722]
  Call Extruder(259.30463)
  MoveL 9834 to (236.39, 160.19, 135.08) mm, rotated rx -180 ry 0 rz -180 deg; joints [-64.505, 66.845, -88.503, 66.097, 99.141, 19.72]
  Call Extruder(260.13252)
  MoveL 9835 to (235.35, 161.1, 135.08) mm, rotated rx -180 ry 0 rz 180 deg; joints [-64.933, 66.879, -88.488, 66.498, 98.977, 19.738]
  Call Extruder(260.29983)
  MoveL 9836 to (235.13, 161.27, 135.08) mm, rotated rx -180 ry 0 rz 180 deg; joints [-65.021, 66.884, -88.486, 66.581, 98.944, 19.745]
  MoveL 9837 to (235.13, 161.27, 135.08) mm, rotated rx -180 ry 0 rz 180 deg; joints [-65.021, 66.884, -88.486, 66.581, 98.944, 19.745]
  Call Extruder(260.63326)
  MoveL 9838 to (234.68, 161.59, 135.08) mm, rotated rx 180 ry 0 rz 180 deg; joints [-65.197, 66.893, -88.482, 66.747, 98.879, 19.758]
  MoveL 9839 to (234.68, 161.59, 135.08) mm, rotated rx 180 ry 0 rz 180 deg; joints [-65.197, 66.893, -88.482, 66.747, 98.879, 19.758]
  Call Extruder(260.96550)
  MoveL 9840 to (234.23, 161.92, 135.08) mm, rotated rx 180 ry 0 rz -180 deg; joints [-65.374, 66.903, -88.478, 66.912, 98.814, 19.771]
  MoveL 9841 to (234.23, 161.92, 135.08) mm, rotated rx 180 ry 0 rz -180 deg; joints [-65.374, 66.903, -88.478, 66.912, 98.814, 19.771]
  Call Extruder(261.08316)
  MoveL 9842 to (234.05, 162.02, 135.08) mm, rotated rx -180 ry 0 rz 180 deg; joints [-65.437, 66.905, -88.477, 66.972, 98.791, 19.778]
  MoveL 9843 to (234.05, 162.02, 135.08) mm, rotated rx -180 ry 0 rz 180 deg; joints [-65.437, 66.905, -88.477, 66.972, 98.791, 19.778]
  Call Extruder(261.29090)
  MoveL 9844 to (233.75, 162.2, 135.08) mm, rotated rx 180 ry 0 rz 180 deg; joints [-65.549, 66.908, -88.475, 67.079, 98.752, 19.79]
  MoveL 9845 to (233.75, 162.2, 135.08) mm, rotated rx 180 ry 0 rz 180 deg; joints [-65.549, 66.908, -88.475, 67.079, 98.752, 19.79]
  Call Extruder(261.49785)
  MoveL 9846 to (233.45, 162.37, 135.08) mm, rotated rx -180 ry 0 rz -180 deg; joints [-65.662, 66.911, -88.474, 67.185, 98.712, 19.802]
  MoveL 9847 to (233.45, 162.37, 135.08) mm, rotated rx -180 ry 0 rz -180 deg; joints [-65.662, 66.911, -88.474, 67.185, 98.712, 19.802]
  Call Extruder(261.70402)
  MoveL 9848 to (233.14, 162.55, 135.08) mm, rotated rx -180 ry 0 rz -180 deg; joints [-65.774, 66.914, -88.473, 67.291, 98.672, 19.814]
  MoveL 9849 to (233.14, 162.55, 135.08) mm, rotated rx -180 ry 0 rz -180 deg; joints [-65.774, 66.914, -88.473, 67.291, 98.672, 19.814]
  Call Extruder(261.88569)
  MoveL 9850 to (232.87, 162.69, 135.08) mm, rotated rx 180 ry 0 rz 180 deg; joints [-65.874, 66.915, -88.472, 67.386, 98.638, 19.826]
  MoveL 9851 to (232.87, 162.69, 135.08) mm, rotated rx 180 ry 0 rz 180 deg; joints [-65.874, 66.915, -88.472, 67.386, 98.638, 19.826]
  Call Extruder(262.04366)
  MoveL 9852 to (232.62, 162.8, 135.08) mm, rotated rx 180 ry 0 rz 180 deg; joints [-65.961, 66.915, -88.472, 67.469, 98.608, 19.839]
  MoveL 9853 to (232.62, 162.8, 135.08) mm, rotated rx 180 ry 0 rz 180 deg; joints [-65.961, 66.915, -88.472, 67.469, 98.608, 19.839]
  Call Extruder(262.20102)
  MoveL 9854 to (232.37, 162.91, 135.08) mm, rotated rx -180 ry 0 rz 180 deg; joints [-66.048, 66.915, -88.472, 67.552, 98.579, 19.852]
  MoveL 9855 to (232.37, 162.91, 135.08) mm, rotated rx -180 ry 0 rz 180 deg; joints [-66.048, 66.915, -88.472, 67.552, 98.579, 19.852]
  Call Extruder(262.38376)
  MoveL 9856 to (232.07, 163.03, 135.08) mm, rotated rx 180 ry 0 rz -180 deg; joints [-66.149, 66.914, -88.473, 67.648, 98.545, 19.868]
  MoveL 9857 to (232.07, 163.03, 135.08) mm, rotated rx 180 ry 0 rz -180 deg; joints [-66.149, 66.914, -88.473, 67.648, 98.545, 19.868]
  Call Extruder(262.56574)
  MoveL 9858 to (231.78, 163.15, 135.08) mm, rotated rx 180 ry 0 rz 180 deg; joints [-66.251, 66.913, -88.473, 67.745, 98.511, 19.883]
  MoveL 9859 to (231.78, 163.15, 135.08) mm, rotated rx 180 ry 0 rz 180 deg; joints [-66.251, 66.913, -88.473, 67.745, 98.511, 19.883]
  Call Extruder(262.71308)
  MoveL 9860 to (231.54, 163.24, 135.08) mm, rotated rx -180 ry 0 rz 180 deg; joints [-66.333, 66.912, -88.474, 67.824, 98.483, 19.896]
  MoveL 9861 to (231.54, 163.24, 135.08) mm, rotated rx -180 ry 0 rz 180 deg; joints [-66.333, 66.912, -88.474, 67.824, 98.483, 19.896]
  Call Extruder(262.82630)
  MoveL 9862 to (231.35, 163.3, 135.08) mm, rotated rx -180 ry 0 rz 180 deg; joints [-66.397, 66.91, -88.474, 67.885, 98.462, 19.907]
  MoveL 9863 to (231.35, 163.3, 135.08) mm, rotated rx -180 ry 0 rz 180 deg; joints [-66.397, 66.91, -88.474, 67.885, 98.462, 19.907]
  Call Extruder(262.93908)
  MoveL 9864 to (231.17, 163.36, 135.08) mm, rotated rx 180 ry 0 rz -180 deg; joints [-66.46, 66.909, -88.475, 67.945, 98.442, 19.918]
  MoveL 9865 to (231.17, 163.36, 135.08) mm, rotated rx 180 ry 0 rz -180 deg; joints [-66.46, 66.909, -88.475, 67.945, 98.442, 19.918]
  Call Extruder(263.05141)
  MoveL 9866 to (230.98, 163.42, 135.08) mm, rotated rx 180 ry 0 rz -180 deg; joints [-66.524, 66.907, -88.476, 68.006, 98.421, 19.93]
  MoveL 9867 to (230.98, 163.42, 135.08) mm, rotated rx 180 ry 0 rz -180 deg; joints [-66.524, 66.907, -88.476, 68.006, 98.421, 19.93]
  Call Extruder(263.16330)
  MoveL 9868 to (230.79, 163.48, 135.08) mm, rotated rx -180 ry 0 rz -180 deg; joints [-66.587, 66.905, -88.477, 68.066, 98.4, 19.941]
  MoveL 9869 to (230.79, 163.48, 135.08) mm, rotated rx -180 ry 0 rz -180 deg; joints [-66.587, 66.905, -88.477, 68.066, 98.4, 19.941]
  Call Extruder(263.28471)
  MoveL 9870 to (230.58, 163.55, 135.08) mm, rotated rx -180 ry 0 rz -180 deg; joints [-66.656, 66.903, -88.477, 68.132, 98.378, 19.953]
  MoveL 9871 to (230.58, 163.55, 135.08) mm, rotated rx -180 ry 0 rz -180 deg; joints [-66.656, 66.903, -88.477, 68.132, 98.378, 19.953]
  Call Extruder(263.41552)
  MoveL 9872 to (230.36, 163.62, 135.08) mm, rotated rx 180 ry 0 rz -180 deg; joints [-66.731, 66.901, -88.478, 68.204, 98.354, 19.966]
  MoveL 9873 to (230.36, 163.62, 135.08) mm, rotated rx 180 ry 0 rz -180 deg; joints [-66.731, 66.901, -88.478, 68.204, 98.354, 19.966]
  Call Extruder(263.54577)
  MoveL 9874 to (230.14, 163.68, 135.08) mm, rotated rx -180 ry 0 rz -180 deg; joints [-66.805, 66.899, -88.48, 68.275, 98.33, 19.98]
  MoveL 9875 to (230.14, 163.68, 135.08) mm, rotated rx -180 ry 0 rz -180 deg; joints [-66.805, 66.899, -88.48, 68.275, 98.33, 19.98]
  Call Extruder(263.67545)
  MoveL 9876 to (229.91, 163.75, 135.08) mm, rotated rx -180 ry 0 rz -180 deg; joints [-66.88, 66.896, -88.481, 68.347, 98.305, 19.993]
  MoveL 9877 to (229.91, 163.75, 135.08) mm, rotated rx -180 ry 0 rz -180 deg; joints [-66.88, 66.896, -88.481, 68.347, 98.305, 19.993]
  Call Extruder(263.80457)
  MoveL 9878 to (229.69, 163.82, 135.08) mm, rotated rx 180 ry 0 rz 180 deg; joints [-66.955, 66.894, -88.482, 68.418, 98.281, 20.007]
  MoveL 9879 to (229.69, 163.82, 135.08) mm, rotated rx 180 ry 0 rz 180 deg; joints [-66.955, 66.894, -88.482, 68.418, 98.281, 20.007]
  Call Extruder(263.91964)
  MoveL 9880 to (229.48, 163.86, 135.08) mm, rotated rx 180 ry 0 rz -180 deg; joints [-67.021, 66.891, -88.483, 68.482, 98.26, 20.02]
  MoveL 9881 to (229.48, 163.86, 135.08) mm, rotated rx 180 ry 0 rz -180 deg; joints [-67.021, 66.891, -88.483, 68.482, 98.26, 20.02]
  Call Extruder(264.03426)
  MoveL 9882 to (229.28, 163.91, 135.08) mm, rotated rx 180 ry 0 rz 180 deg; joints [-67.087, 66.887, -88.485, 68.545, 98.239, 20.034]
  MoveL 9883 to (229.28, 163.91, 135.08) mm, rotated rx 180 ry 0 rz 180 deg; joints [-67.087, 66.887, -88.485, 68.545, 98.239, 20.034]
  Call Extruder(264.14843)
  MoveL 9884 to (229.08, 163.95, 135.08) mm, rotated rx -180 ry 0 rz 180 deg; joints [-67.153, 66.884, -88.486, 68.608, 98.218, 20.048]
  MoveL 9885 to (229.08, 163.95, 135.08) mm, rotated rx -180 ry 0 rz 180 deg; joints [-67.153, 66.884, -88.486, 68.608, 98.218, 20.048]
  Call Extruder(264.26215)
  MoveL 9886 to (228.87, 164, 135.08) mm, rotated rx -180 ry 0 rz -180 deg; joints [-67.22, 66.88, -88.488, 68.672, 98.197, 20.061]
  MoveL 9887 to (228.87, 164, 135.08) mm, rotated rx -180 ry 0 rz -180 deg; joints [-67.22, 66.88, -88.488, 68.672, 98.197, 20.061]
  Call Extruder(264.38757)
  MoveL 9888 to (228.64, 164.04, 135.08) mm, rotated rx 180 ry 0 rz -180 deg; joints [-67.293, 66.876, -88.489, 68.742, 98.174, 20.077]
  MoveL 9889 to (228.64, 164.04, 135.08) mm, rotated rx 180 ry 0 rz -180 deg; joints [-67.293, 66.876, -88.489, 68.742, 98.174, 20.077]
  Call Extruder(264.52455)
  MoveL 9890 to (228.4, 164.09, 135.08) mm, rotated rx -180 ry 0 rz 180 deg; joints [-67.373, 66.872, -88.491, 68.819, 98.149, 20.093]
  MoveL 9891 to (228.4, 164.09, 135.08) mm, rotated rx -180 ry 0 rz 180 deg; joints [-67.373, 66.872, -88.491, 68.819, 98.149, 20.093]
  Call Extruder(264.66091)
  MoveL 9892 to (228.15, 164.14, 135.08) mm, rotated rx -180 ry 0 rz 180 deg; joints [-67.453, 66.867, -88.493, 68.896, 98.124, 20.11]
  MoveL 9893 to (228.15, 164.14, 135.08) mm, rotated rx -180 ry 0 rz 180 deg; joints [-67.453, 66.867, -88.493, 68.896, 98.124, 20.11]
  Call Extruder(264.79667)
  MoveL 9894 to (227.9, 164.19, 135.08) mm, rotated rx -180 ry 0 rz -180 deg; joints [-67.534, 66.863, -88.495, 68.973, 98.099, 20.127]
  MoveL 9895 to (227.9, 164.19, 135.08) mm, rotated rx -180 ry 0 rz -180 deg; joints [-67.534, 66.863, -88.495, 68.973, 98.099, 20.127]
  Call Extruder(264.93182)
  MoveL 9896 to (227.65, 164.24, 135.08) mm, rotated rx -180 ry 0 rz 180 deg; joints [-67.614, 66.858, -88.497, 69.05, 98.073, 20.144]
  MoveL 9897 to (227.65, 164.24, 135.08) mm, rotated rx -180 ry 0 rz 180 deg; joints [-67.614, 66.858, -88.497, 69.05, 98.073, 20.144]
  Call Extruder(265.06636)
  MoveL 9898 to (227.4, 164.29, 135.08) mm, rotated rx 180 ry 0 rz 180 deg; joints [-67.695, 66.854, -88.499, 69.127, 98.048, 20.161]
  MoveL 9899 to (227.4, 164.29, 135.08) mm, rotated rx 180 ry 0 rz 180 deg; joints [-67.695, 66.854, -88.499, 69.127, 98.048, 20.161]
  Call Extruder(265.20028)
  MoveL 9900 to (227.15, 164.34, 135.08) mm, rotated rx -180 ry 0 rz 180 deg; joints [-67.775, 66.85, -88.501, 69.204, 98.022, 20.177]
  MoveL 9901 to (227.15, 164.34, 135.08) mm, rotated rx -180 ry 0 rz 180 deg; joints [-67.775, 66.85, -88.501, 69.204, 98.022, 20.177]
  Call Extruder(265.34815)
  MoveL 9902 to (226.87, 164.39, 135.08) mm, rotated rx -180 ry 0 rz 180 deg; joints [-67.864, 66.844, -88.503, 69.29, 97.994, 20.196]
  MoveL 9903 to (226.87, 164.39, 135.08) mm, rotated rx -180 ry 0 rz 180 deg; joints [-67.864, 66.844, -88.503, 69.29, 97.994, 20.196]
  Call Extruder(265.50989)
  MoveL 9904 to (226.57, 164.44, 135.08) mm, rotated rx 180 ry 0 rz 180 deg; joints [-67.961, 66.838, -88.506, 69.383, 97.964, 20.217]
  MoveL 9905 to (226.57, 164.44, 135.08) mm, rotated rx 180 ry 0 rz 180 deg; joints [-67.961, 66.838, -88.506, 69.383, 97.964, 20.217]
  Call Extruder(265.67090)
  MoveL 9906 to (226.26, 164.49, 135.08) mm, rotated rx 180 ry 0 rz 180 deg; joints [-68.059, 66.832, -88.509, 69.477, 97.933, 20.239]
  MoveL 9907 to (226.26, 164.49, 135.08) mm, rotated rx 180 ry 0 rz 180 deg; joints [-68.059, 66.832, -88.509, 69.477, 97.933, 20.239]
  Call Extruder(265.83118)
  MoveL 9908 to (225.95, 164.54, 135.08) mm, rotated rx 180 ry 0 rz -180 deg; joints [-68.156, 66.826, -88.512, 69.57, 97.903, 20.26]
  MoveL 9909 to (225.95, 164.54, 135.08) mm, rotated rx 180 ry 0 rz -180 deg; joints [-68.156, 66.826, -88.512, 69.57, 97.903, 20.26]
  Call Extruder(265.99074)
  MoveL 9910 to (225.65, 164.58, 135.08) mm, rotated rx 180 ry 0 rz 180 deg; joints [-68.254, 66.819, -88.514, 69.664, 97.872, 20.281]
  MoveL 9911 to (225.65, 164.58, 135.08) mm, rotated rx 180 ry 0 rz 180 deg; joints [-68.254, 66.819, -88.514, 69.664, 97.872, 20.281]
  Call Extruder(266.14957)
  MoveL 9912 to (225.34, 164.63, 135.08) mm, rotated rx -180 ry 0 rz 180 deg; joints [-68.351, 66.813, -88.517, 69.757, 97.841, 20.302]
  MoveL 9913 to (225.34, 164.63, 135.08) mm, rotated rx -180 ry 0 rz 180 deg; joints [-68.351, 66.813, -88.517, 69.757, 97.841, 20.302]
  Call Extruder(266.32824)
  MoveL 9914 to (225, 164.68, 135.08) mm, rotated rx -180 ry 0 rz 180 deg; joints [-68.461, 66.806, -88.52, 69.863, 97.807, 20.326]
  MoveL 9915 to (225, 164.68, 135.08) mm, rotated rx -180 ry 0 rz 180 deg; joints [-68.461, 66.806, -88.52, 69.863, 97.807, 20.326]
  Call Extruder(266.52668)
  MoveL 9916 to (224.61, 164.72, 135.08) mm, rotated rx -180 ry 0 rz 180 deg; joints [-68.583, 66.797, -88.524, 69.98, 97.769, 20.354]
  MoveL 9917 to (224.61, 164.72, 135.08) mm, rotated rx -180 ry 0 rz 180 deg; joints [-68.583, 66.797, -88.524, 69.98, 97.769, 20.354]
  Call Extruder(266.72426)
  MoveL 9918 to (224.22, 164.77, 135.08) mm, rotated rx -180 ry 0 rz 180 deg; joints [-68.706, 66.788, -88.528, 70.098, 97.73, 20.382]
  MoveL 9919 to (224.22, 164.77, 135.08) mm, rotated rx -180 ry 0 rz 180 deg; joints [-68.706, 66.788, -88.528, 70.098, 97.73, 20.382]
  Call Extruder(266.92097)
  MoveL 9920 to (223.84, 164.82, 135.08) mm, rotated rx 180 ry 0 rz 180 deg; joints [-68.828, 66.779, -88.532, 70.215, 97.692, 20.409]
  MoveL 9921 to (223.84, 164.82, 135.08) mm, rotated rx 180 ry 0 rz 180 deg; joints [-68.828, 66.779, -88.532, 70.215, 97.692, 20.409]
  Call Extruder(267.11680)
  MoveL 9922 to (223.45, 164.86, 135.08) mm, rotated rx -180 ry 0 rz 180 deg; joints [-68.951, 66.77, -88.536, 70.332, 97.654, 20.437]
  MoveL 9923 to (223.45, 164.86, 135.08) mm, rotated rx -180 ry 0 rz 180 deg; joints [-68.951, 66.77, -88.536, 70.332, 97.654, 20.437]
  Call Extruder(267.41216)
  MoveL 9924 to (222.86, 164.91, 135.08) mm, rotated rx -180 ry 0 rz 180 deg; joints [-69.135, 66.755, -88.542, 70.509, 97.596, 20.48]
  MoveL 9925 to (222.86, 164.91, 135.08) mm, rotated rx -180 ry 0 rz 180 deg; joints [-69.135, 66.755, -88.542, 70.509, 97.596, 20.48]
  Call Extruder(267.70619)
  MoveL 9926 to (222.27, 164.96, 135.08) mm, rotated rx -180 ry 0 rz 180 deg; joints [-69.319, 66.74, -88.549, 70.686, 97.539, 20.524]
  MoveL 9927 to (222.27, 164.96, 135.08) mm, rotated rx -180 ry 0 rz 180 deg; joints [-69.319, 66.74, -88.549, 70.686, 97.539, 20.524]
  Call Extruder(267.99889)
  MoveL 9928 to (221.68, 165, 135.08) mm, rotated rx -180 ry 0 rz 180 deg; joints [-69.504, 66.726, -88.555, 70.863, 97.481, 20.567]
  MoveL 9929 to (221.68, 165, 135.08) mm, rotated rx -180 ry 0 rz 180 deg; joints [-69.504, 66.726, -88.555, 70.863, 97.481, 20.567]
  Call Extruder(268.57233)
  MoveL 9930 to (220.52, 165.05, 135.08) mm, rotated rx -180 ry 0 rz 180 deg; joints [-69.864, 66.693, -88.569, 71.209, 97.37, 20.655]
  MoveL 9931 to (220.52, 165.05, 135.08) mm, rotated rx -180 ry 0 rz 180 deg; joints [-69.864, 66.693, -88.569, 71.209, 97.37, 20.655]
  Call Extruder(269.28634)
  MoveL 9932 to (219.06, 165.09, 135.08) mm, rotated rx -180 ry 0 rz -180 deg; joints [-70.315, 66.652, -88.587, 71.641, 97.229, 20.766]
  Call Extruder(386.13307)
  MoveL 9933 to (-19.06, 165.09, 135.08) mm, rotated rx -180 ry 0 rz 180 deg; joints [-137.325, 72.079, -85.07, 136.584, 80.487, 8.888]
  Call Extruder(386.56168)
  MoveL 9934 to (-19.94, 165.07, 135.08) mm, rotated rx 180 ry 0 rz 180 deg; joints [-137.467, 72.122, -85.029, 136.736, 80.526, 8.806]
  MoveL 9935 to (-19.94, 165.07, 135.08) mm, rotated rx 180 ry 0 rz 180 deg; joints [-137.467, 72.122, -85.029, 136.736, 80.526, 8.806]
  Call Extruder(387.13513)
  MoveL 9936 to (-21.1, 165.02, 135.08) mm, rotated rx 180 ry 0 rz 180 deg; joints [-137.659, 72.178, -84.975, 136.94, 80.577, 8.699]
  MoveL 9937 to (-21.1, 165.02, 135.08) mm, rotated rx 180 ry 0 rz 180 deg; joints [-137.659, 72.178, -84.975, 136.94, 80.577, 8.699]
  Call Extruder(387.56943)
  MoveL 9938 to (-21.97, 164.98, 135.08) mm, rotated rx -180 ry 0 rz 180 deg; joints [-137.804, 72.22, -84.935, 137.096, 80.615, 8.618]
  MoveL 9939 to (-21.97, 164.98, 135.08) mm, rotated rx -180 ry 0 rz 180 deg; joints [-137.804, 72.22, -84.935, 137.096, 80.615, 8.618]
  Call Extruder(387.86345)
  MoveL 9940 to (-22.56, 164.93, 135.08) mm, rotated rx -180 ry 0 rz 180 deg; joints [-137.905, 72.247, -84.909, 137.202, 80.639, 8.565]
  MoveL 9941 to (-22.56, 164.93, 135.08) mm, rotated rx -180 ry 0 rz 180 deg; joints [-137.905, 72.247, -84.909, 137.202, 80.639, 8.565]
  Call Extruder(388.15881)
  MoveL 9942 to (-23.15, 164.89, 135.08) mm, rotated rx -180 ry 0 rz -180 deg; joints [-138.004, 72.274, -84.882, 137.308, 80.664, 8.511]
  MoveL 9943 to (-23.15, 164.89, 135.08) mm, rotated rx -180 ry 0 rz -180 deg; joints [-138.004, 72.274, -84.882, 137.308, 80.664, 8.511]
  Call Extruder(388.40503)
  MoveL 9944 to (-23.64, 164.84, 135.08) mm, rotated rx -180 ry 0 rz -180 deg; joints [-138.088, 72.297, -84.86, 137.397, 80.684, 8.467]
  MoveL 9945 to (-23.64, 164.84, 135.08) mm, rotated rx -180 ry 0 rz -180 deg; joints [-138.088, 72.297, -84.86, 137.397, 80.684, 8.467]
  Call Extruder(388.60173)
  MoveL 9946 to (-24.03, 164.79, 135.08) mm, rotated rx 180 ry 0 rz 180 deg; joints [-138.156, 72.314, -84.844, 137.469, 80.699, 8.433]
  MoveL 9947 to (-24.03, 164.79, 135.08) mm, rotated rx 180 ry 0 rz 180 deg; joints [-138.156, 72.314, -84.844, 137.469, 80.699, 8.433]
  Call Extruder(388.79931)
  MoveL 9948 to (-24.42, 164.75, 135.08) mm, rotated rx -180 ry 0 rz 180 deg; joints [-138.224, 72.331, -84.827, 137.541, 80.715, 8.399]
  MoveL 9949 to (-24.42, 164.75, 135.08) mm, rotated rx -180 ry 0 rz 180 deg; joints [-138.224, 72.331, -84.827, 137.541, 80.715, 8.399]
  Call Extruder(388.99775)
  MoveL 9950 to (-24.8, 164.7, 135.08) mm, rotated rx 180 ry 0 rz 180 deg; joints [-138.292, 72.349, -84.81, 137.612, 80.73, 8.364]
  MoveL 9951 to (-24.8, 164.7, 135.08) mm, rotated rx 180 ry 0 rz 180 deg; joints [-138.292, 72.349, -84.81, 137.612, 80.73, 8.364]
  Call Extruder(389.19706)
  MoveL 9952 to (-25.19, 164.66, 135.08) mm, rotated rx 180 ry 0 rz 180 deg; joints [-138.359, 72.366, -84.793, 137.684, 80.746, 8.33]
  MoveL 9953 to (-25.19, 164.66, 135.08) mm, rotated rx 180 ry 0 rz 180 deg; joints [-138.359, 72.366, -84.793, 137.684, 80.746, 8.33]
  Call Extruder(389.35589)
  MoveL 9954 to (-25.5, 164.61, 135.08) mm, rotated rx -180 ry 0 rz 180 deg; joints [-138.415, 72.379, -84.78, 137.742, 80.757, 8.303]
  MoveL 9955 to (-25.5, 164.61, 135.08) mm, rotated rx -180 ry 0 rz 180 deg; joints [-138.415, 72.379, -84.78, 137.742, 80.757, 8.303]
  Call Extruder(389.51545)
  MoveL 9956 to (-25.8, 164.56, 135.08) mm, rotated rx -180 ry 0 rz 180 deg; joints [-138.47, 72.392, -84.767, 137.8, 80.768, 8.276]
  MoveL 9957 to (-25.8, 164.56, 135.08) mm, rotated rx -180 ry 0 rz 180 deg; joints [-138.47, 72.392, -84.767, 137.8, 80.768, 8.276]
  Call Extruder(389.67574)
  MoveL 9958 to (-26.11, 164.51, 135.08) mm, rotated rx -180 ry 0 rz 180 deg; joints [-138.525, 72.405, -84.754, 137.858, 80.78, 8.25]
  MoveL 9959 to (-26.11, 164.51, 135.08) mm, rotated rx -180 ry 0 rz 180 deg; joints [-138.525, 72.405, -84.754, 137.858, 80.78, 8.25]
  Call Extruder(389.83676)
  MoveL 9960 to (-26.41, 164.46, 135.08) mm, rotated rx -180 ry 0 rz 180 deg; joints [-138.58, 72.418, -84.741, 137.917, 80.791, 8.223]
  MoveL 9961 to (-26.41, 164.46, 135.08) mm, rotated rx -180 ry 0 rz 180 deg; joints [-138.58, 72.418, -84.741, 137.917, 80.791, 8.223]
  Call Extruder(389.99850)
  MoveL 9962 to (-26.72, 164.41, 135.08) mm, rotated rx -180 ry 0 rz 180 deg; joints [-138.635, 72.431, -84.727, 137.974, 80.803, 8.197]
  MoveL 9963 to (-26.72, 164.41, 135.08) mm, rotated rx -180 ry 0 rz 180 deg; joints [-138.635, 72.431, -84.727, 137.974, 80.803, 8.197]
  Call Extruder(390.16097)
  MoveL 9964 to (-27.03, 164.37, 135.08) mm, rotated rx 180 ry 0 rz -180 deg; joints [-138.69, 72.445, -84.714, 138.032, 80.815, 8.17]
  MoveL 9965 to (-27.03, 164.37, 135.08) mm, rotated rx 180 ry 0 rz -180 deg; joints [-138.69, 72.445, -84.714, 138.032, 80.815, 8.17]
  Call Extruder(390.29490)
  MoveL 9966 to (-27.27, 164.32, 135.08) mm, rotated rx -180 ry 0 rz -180 deg; joints [-138.736, 72.455, -84.704, 138.081, 80.823, 8.149]
  MoveL 9967 to (-27.27, 164.32, 135.08) mm, rotated rx -180 ry 0 rz -180 deg; joints [-138.736, 72.455, -84.704, 138.081, 80.823, 8.149]
  Call Extruder(390.42943)
  MoveL 9968 to (-27.52, 164.27, 135.08) mm, rotated rx -180 ry 0 rz 180 deg; joints [-138.783, 72.465, -84.694, 138.13, 80.832, 8.127]
  MoveL 9969 to (-27.52, 164.27, 135.08) mm, rotated rx -180 ry 0 rz 180 deg; joints [-138.783, 72.465, -84.694, 138.13, 80.832, 8.127]
  Call Extruder(390.56458)
  MoveL 9970 to (-27.77, 164.22, 135.08) mm, rotated rx -180 ry 0 rz 180 deg; joints [-138.829, 72.475, -84.684, 138.178, 80.841, 8.106]
  MoveL 9971 to (-27.77, 164.22, 135.08) mm, rotated rx -180 ry 0 rz 180 deg; joints [-138.829, 72.475, -84.684, 138.178, 80.841, 8.106]
  Call Extruder(390.70034)
  MoveL 9972 to (-28.02, 164.17, 135.08) mm, rotated rx -180 ry 0 rz -180 deg; joints [-138.875, 72.486, -84.673, 138.227, 80.85, 8.085]
  MoveL 9973 to (-28.02, 164.17, 135.08) mm, rotated rx -180 ry 0 rz -180 deg; joints [-138.875, 72.486, -84.673, 138.227, 80.85, 8.085]
  Call Extruder(390.83670)
  MoveL 9974 to (-28.27, 164.12, 135.08) mm, rotated rx -180 ry 0 rz -180 deg; joints [-138.921, 72.496, -84.663, 138.275, 80.858, 8.064]
  MoveL 9975 to (-28.27, 164.12, 135.08) mm, rotated rx -180 ry 0 rz -180 deg; joints [-138.921, 72.496, -84.663, 138.275, 80.858, 8.064]
  Call Extruder(390.97368)
  MoveL 9976 to (-28.52, 164.07, 135.08) mm, rotated rx 180 ry 0 rz 180 deg; joints [-138.967, 72.506, -84.653, 138.324, 80.867, 8.042]
  MoveL 9977 to (-28.52, 164.07, 135.08) mm, rotated rx 180 ry 0 rz 180 deg; joints [-138.967, 72.506, -84.653, 138.324, 80.867, 8.042]
  Call Extruder(391.11127)
  MoveL 9978 to (-28.77, 164.02, 135.08) mm, rotated rx -180 ry 0 rz 180 deg; joints [-139.013, 72.516, -84.642, 138.372, 80.876, 8.021]
  MoveL 9979 to (-28.77, 164.02, 135.08) mm, rotated rx -180 ry 0 rz 180 deg; joints [-139.013, 72.516, -84.642, 138.372, 80.876, 8.021]
  Call Extruder(391.22498)
  MoveL 9980 to (-28.97, 163.97, 135.08) mm, rotated rx -180 ry 0 rz 180 deg; joints [-139.052, 72.525, -84.634, 138.412, 80.883, 8.004]
  MoveL 9981 to (-28.97, 163.97, 135.08) mm, rotated rx -180 ry 0 rz 180 deg; joints [-139.052, 72.525, -84.634, 138.412, 80.883, 8.004]
  Call Extruder(391.33915)
  MoveL 9982 to (-29.18, 163.93, 135.08) mm, rotated rx 180 ry 0 rz 180 deg; joints [-139.09, 72.533, -84.625, 138.453, 80.89, 7.987]
  MoveL 9983 to (-29.18, 163.93, 135.08) mm, rotated rx 180 ry 0 rz 180 deg; joints [-139.09, 72.533, -84.625, 138.453, 80.89, 7.987]
  Call Extruder(391.45377)
  MoveL 9984 to (-29.38, 163.88, 135.08) mm, rotated rx -180 ry 0 rz 180 deg; joints [-139.128, 72.541, -84.617, 138.493, 80.898, 7.97]
  MoveL 9985 to (-29.38, 163.88, 135.08) mm, rotated rx -180 ry 0 rz 180 deg; joints [-139.128, 72.541, -84.617, 138.493, 80.898, 7.97]
  Call Extruder(391.56884)
  MoveL 9986 to (-29.59, 163.84, 135.08) mm, rotated rx 180 ry 0 rz 180 deg; joints [-139.166, 72.549, -84.609, 138.533, 80.905, 7.952]
  MoveL 9987 to (-29.59, 163.84, 135.08) mm, rotated rx 180 ry 0 rz 180 deg; joints [-139.166, 72.549, -84.609, 138.533, 80.905, 7.952]
  Call Extruder(391.69108)
  MoveL 9988 to (-29.8, 163.78, 135.08) mm, rotated rx -180 ry 0 rz 180 deg; joints [-139.208, 72.558, -84.6, 138.576, 80.911, 7.935]
  MoveL 9989 to (-29.8, 163.78, 135.08) mm, rotated rx -180 ry 0 rz 180 deg; joints [-139.208, 72.558, -84.6, 138.576, 80.911, 7.935]
  Call Extruder(391.82075)
  MoveL 9990 to (-30.02, 163.72, 135.08) mm, rotated rx -180 ry 0 rz 180 deg; joints [-139.253, 72.566, -84.592, 138.624, 80.918, 7.916]
  MoveL 9991 to (-30.02, 163.72, 135.08) mm, rotated rx -180 ry 0 rz 180 deg; joints [-139.253, 72.566, -84.592, 138.624, 80.918, 7.916]
  Call Extruder(391.95100)
  MoveL 9992 to (-30.25, 163.65, 135.08) mm, rotated rx -180 ry 0 rz -180 deg; joints [-139.298, 72.574, -84.584, 138.67, 80.924, 7.898]
  MoveL 9993 to (-30.25, 163.65, 135.08) mm, rotated rx -180 ry 0 rz -180 deg; joints [-139.298, 72.574, -84.584, 138.67, 80.924, 7.898]
  Call Extruder(392.08180)
  MoveL 9994 to (-30.47, 163.58, 135.08) mm, rotated rx -180 ry 0 rz 180 deg; joints [-139.343, 72.582, -84.575, 138.717, 80.93, 7.88]
  MoveL 9995 to (-30.47, 163.58, 135.08) mm, rotated rx -180 ry 0 rz 180 deg; joints [-139.343, 72.582, -84.575, 138.717, 80.93, 7.88]
  Call Extruder(392.21318)
  MoveL 9996 to (-30.7, 163.51, 135.08) mm, rotated rx 180 ry 0 rz 180 deg; joints [-139.388, 72.591, -84.567, 138.764, 80.937, 7.861]
  MoveL 9997 to (-30.7, 163.51, 135.08) mm, rotated rx 180 ry 0 rz 180 deg; joints [-139.388, 72.591, -84.567, 138.764, 80.937, 7.861]
  Call Extruder(392.32507)
  MoveL 9998 to (-30.88, 163.45, 135.08) mm, rotated rx -180 ry 0 rz 180 deg; joints [-139.427, 72.597, -84.56, 138.804, 80.942, 7.846]
  MoveL 9999 to (-30.88, 163.45, 135.08) mm, rotated rx -180 ry 0 rz 180 deg; joints [-139.427, 72.597, -84.56, 138.804, 80.942, 7.846]
  Call Extruder(392.43740)
  MoveL 10000 to (-31.07, 163.39, 135.08) mm, rotated rx 180 ry 0 rz -180 deg; joints [-139.465, 72.604, -84.553, 138.844, 80.947, 7.831]
  MoveL 10001 to (-31.07, 163.39, 135.08) mm, rotated rx 180 ry 0 rz -180 deg; joints [-139.465, 72.604, -84.553, 138.844, 80.947, 7.831]
  Call Extruder(392.55019)
  MoveL 10002 to (-31.26, 163.33, 135.08) mm, rotated rx -180 ry 0 rz 180 deg; joints [-139.504, 72.611, -84.546, 138.885, 80.952, 7.816]
  MoveL 10003 to (-31.26, 163.33, 135.08) mm, rotated rx -180 ry 0 rz 180 deg; joints [-139.504, 72.611, -84.546, 138.885, 80.952, 7.816]
  Call Extruder(392.66341)
  MoveL 10004 to (-31.45, 163.27, 135.08) mm, rotated rx 180 ry 0 rz -180 deg; joints [-139.542, 72.618, -84.539, 138.925, 80.957, 7.801]
  MoveL 10005 to (-31.45, 163.27, 135.08) mm, rotated rx 180 ry 0 rz -180 deg; joints [-139.542, 72.618, -84.539, 138.925, 80.957, 7.801]
  Call Extruder(392.77708)
  MoveL 10006 to (-31.64, 163.21, 135.08) mm, rotated rx -180 ry 0 rz 180 deg; joints [-139.581, 72.624, -84.532, 138.964, 80.962, 7.785]
  MoveL 10007 to (-31.64, 163.21, 135.08) mm, rotated rx -180 ry 0 rz 180 deg; joints [-139.581, 72.624, -84.532, 138.964, 80.962, 7.785]
  Call Extruder(392.95906)
  MoveL 10008 to (-31.93, 163.09, 135.08) mm, rotated rx 180 ry 0 rz 180 deg; joints [-139.645, 72.634, -84.522, 139.031, 80.968, 7.763]
  MoveL 10009 to (-31.93, 163.09, 135.08) mm, rotated rx 180 ry 0 rz 180 deg; joints [-139.645, 72.634, -84.522, 139.031, 80.968, 7.763]
  Call Extruder(393.14179)
  MoveL 10010 to (-32.22, 162.96, 135.08) mm, rotated rx -180 ry 0 rz -180 deg; joints [-139.709, 72.643, -84.512, 139.097, 80.974, 7.74]
  MoveL 10011 to (-32.22, 162.96, 135.08) mm, rotated rx -180 ry 0 rz -180 deg; joints [-139.709, 72.643, -84.512, 139.097, 80.974, 7.74]
  Call Extruder(393.31221)
  MoveL 10012 to (-32.49, 162.85, 135.08) mm, rotated rx -180 ry 0 rz 180 deg; joints [-139.768, 72.652, -84.503, 139.158, 80.979, 7.719]
  MoveL 10013 to (-32.49, 162.85, 135.08) mm, rotated rx -180 ry 0 rz 180 deg; joints [-139.768, 72.652, -84.503, 139.158, 80.979, 7.719]
  Call Extruder(393.47018)
  MoveL 10014 to (-32.74, 162.74, 135.08) mm, rotated rx -180 ry 0 rz -180 deg; joints [-139.823, 72.66, -84.495, 139.215, 80.984, 7.699]
  MoveL 10015 to (-32.74, 162.74, 135.08) mm, rotated rx -180 ry 0 rz -180 deg; joints [-139.823, 72.66, -84.495, 139.215, 80.984, 7.699]
  Call Extruder(393.62876)
  MoveL 10016 to (-32.99, 162.64, 135.08) mm, rotated rx 180 ry 0 rz 180 deg; joints [-139.878, 72.668, -84.487, 139.272, 80.989, 7.68]
  MoveL 10017 to (-32.99, 162.64, 135.08) mm, rotated rx 180 ry 0 rz 180 deg; joints [-139.878, 72.668, -84.487, 139.272, 80.989, 7.68]
  Call Extruder(393.83493)
  MoveL 10018 to (-33.29, 162.46, 135.08) mm, rotated rx 180 ry 0 rz 180 deg; joints [-139.953, 72.676, -84.479, 139.349, 80.991, 7.658]
  MoveL 10019 to (-33.29, 162.46, 135.08) mm, rotated rx 180 ry 0 rz 180 deg; joints [-139.953, 72.676, -84.479, 139.349, 80.991, 7.658]
  Call Extruder(394.04187)
  MoveL 10020 to (-33.6, 162.29, 135.08) mm, rotated rx -180 ry 0 rz 180 deg; joints [-140.028, 72.683, -84.471, 139.426, 80.993, 7.636]
  MoveL 10021 to (-33.6, 162.29, 135.08) mm, rotated rx -180 ry 0 rz 180 deg; joints [-140.028, 72.683, -84.471, 139.426, 80.993, 7.636]
  Call Extruder(394.24959)
  MoveL 10022 to (-33.9, 162.11, 135.08) mm, rotated rx -180 ry 0 rz -180 deg; joints [-140.103, 72.691, -84.463, 139.502, 80.995, 7.613]
  MoveL 10023 to (-33.9, 162.11, 135.08) mm, rotated rx -180 ry 0 rz -180 deg; joints [-140.103, 72.691, -84.463, 139.502, 80.995, 7.613]
  Call Extruder(394.45809)
  MoveL 10024 to (-34.21, 161.94, 135.08) mm, rotated rx -180 ry 0 rz 180 deg; joints [-140.178, 72.699, -84.454, 139.579, 80.998, 7.591]
  MoveL 10025 to (-34.21, 161.94, 135.08) mm, rotated rx -180 ry 0 rz 180 deg; joints [-140.178, 72.699, -84.454, 139.579, 80.998, 7.591]
  Call Extruder(394.63764)
  MoveL 10026 to (-34.45, 161.76, 135.08) mm, rotated rx 180 ry 0 rz 180 deg; joints [-140.244, 72.704, -84.449, 139.647, 80.997, 7.574]
  MoveL 10027 to (-34.45, 161.76, 135.08) mm, rotated rx 180 ry 0 rz 180 deg; joints [-140.244, 72.704, -84.449, 139.647, 80.997, 7.574]
  Call Extruder(394.97107)
  MoveL 10028 to (-34.9, 161.43, 135.08) mm, rotated rx -180 ry 0 rz 180 deg; joints [-140.366, 72.713, -84.44, 139.771, 80.994, 7.543]
  MoveL 10029 to (-34.9, 161.43, 135.08) mm, rotated rx -180 ry 0 rz 180 deg; joints [-140.366, 72.713, -84.44, 139.771, 80.994, 7.543]
  Call Extruder(395.30569)
  MoveL 10030 to (-35.35, 161.1, 135.08) mm, rotated rx -180 ry 0 rz -180 deg; joints [-140.489, 72.722, -84.431, 139.896, 80.993, 7.511]
  Call Extruder(396.13360)
  MoveL 10031 to (-36.39, 160.19, 135.08) mm, rotated rx 180 ry 0 rz 180 deg; joints [-140.797, 72.737, -84.415, 140.209, 80.975, 7.444]
  Call Extruder(396.96153)
  MoveL 10032 to (-37.3, 159.15, 135.08) mm, rotated rx 180 ry 0 rz 180 deg; joints [-141.109, 72.74, -84.412, 140.522, 80.941, 7.39]
  Call Extruder(397.12884)
  MoveL 10033 to (-37.47, 158.93, 135.08) mm, rotated rx -180 ry 0 rz -180 deg; joints [-141.172, 72.739, -84.413, 140.586, 80.931, 7.381]
  MoveL 10034 to (-37.47, 158.93, 135.08) mm, rotated rx -180 ry 0 rz -180 deg; joints [-141.172, 72.739, -84.413, 140.586, 80.931, 7.381]
  Call Extruder(397.46227)
  MoveL 10035 to (-37.79, 158.48, 135.08) mm, rotated rx -180 ry 0 rz -180 deg; joints [-141.298, 72.737, -84.414, 140.712, 80.912, 7.363]
  MoveL 10036 to (-37.79, 158.48, 135.08) mm, rotated rx -180 ry 0 rz -180 deg; joints [-141.298, 72.737, -84.414, 140.712, 80.912, 7.363]
  Call Extruder(397.53291)
  MoveL 10037 to (-37.86, 158.38, 135.08) mm, rotated rx -180 ry 0 rz -180 deg; joints [-141.324, 72.737, -84.415, 140.739, 80.908, 7.359]
  Set speed (130.0 mm/s)
  MoveL 10038 to (-39.48, 155.51, 135.08) mm, rotated rx 180 ry 0 rz -180 deg; joints [-142.061, 72.704, -84.45, 141.472, 80.761, 7.285]
  MoveL 10039 to (-39.48, 155.51, 144.49) mm, rotated rx -180 ry 0 rz -180 deg; joints [-142.061, 74.06, -86.181, 141.433, 80.468, 7.522]
  MoveL 10040 to (-38.84, 156.79, 144.49) mm, rotated rx -180 ry 0 rz -180 deg; joints [-141.743, 74.079, -86.162, 141.117, 80.539, 7.55]
  Set speed (30.0 mm/s)
  MoveL 10041 to (-38.84, 156.79, 144.49) mm, rotated rx -180 ry 0 rz -180 deg; joints [-141.743, 74.079, -86.162, 141.117, 80.539, 7.55]
  Call Extruder(397.61221)
  MoveL 10042 to (-38.89, 156.67, 144.49) mm, rotated rx 180 ry 0 rz -180 deg; joints [-141.773, 74.077, -86.164, 141.147, 80.532, 7.548]
  MoveL 10043 to (-38.89, 156.67, 144.49) mm, rotated rx 180 ry 0 rz -180 deg; joints [-141.773, 74.077, -86.164, 141.147, 80.532, 7.548]
  Call Extruder(397.77019)
  MoveL 10044 to (-39, 156.42, 144.49) mm, rotated rx -180 ry 0 rz 180 deg; joints [-141.832, 74.072, -86.169, 141.205, 80.517, 7.545]
  MoveL 10045 to (-39, 156.42, 144.49) mm, rotated rx -180 ry 0 rz 180 deg; joints [-141.832, 74.072, -86.169, 141.205, 80.517, 7.545]
  Call Extruder(397.92758)
  MoveL 10046 to (-39.1, 156.17, 144.49) mm, rotated rx -180 ry 0 rz 180 deg; joints [-141.891, 74.068, -86.174, 141.264, 80.502, 7.541]
  MoveL 10047 to (-39.1, 156.17, 144.49) mm, rotated rx -180 ry 0 rz 180 deg; joints [-141.891, 74.068, -86.174, 141.264, 80.502, 7.541]
  Call Extruder(398.11030)
  MoveL 10048 to (-39.23, 155.88, 144.49) mm, rotated rx 180 ry 0 rz 180 deg; joints [-141.96, 74.062, -86.179, 141.332, 80.484, 7.537]
  MoveL 10049 to (-39.23, 155.88, 144.49) mm, rotated rx 180 ry 0 rz 180 deg; joints [-141.96, 74.062, -86.179, 141.332, 80.484, 7.537]
  Call Extruder(398.29226)
  MoveL 10050 to (-39.35, 155.58, 144.49) mm, rotated rx 180 ry 0 rz 180 deg; joints [-142.029, 74.056, -86.185, 141.4, 80.466, 7.532]
  MoveL 10051 to (-39.35, 155.58, 144.49) mm, rotated rx 180 ry 0 rz 180 deg; joints [-142.029, 74.056, -86.185, 141.4, 80.466, 7.532]
  Call Extruder(398.43959)
  MoveL 10052 to (-39.44, 155.34, 144.49) mm, rotated rx -180 ry 0 rz 180 deg; joints [-142.085, 74.051, -86.19, 141.455, 80.451, 7.529]
  MoveL 10053 to (-39.44, 155.34, 144.49) mm, rotated rx -180 ry 0 rz 180 deg; joints [-142.085, 74.051, -86.19, 141.455, 80.451, 7.529]
  Call Extruder(398.55283)
  MoveL 10054 to (-39.5, 155.15, 144.49) mm, rotated rx -180 ry 0 rz 180 deg; joints [-142.127, 74.047, -86.195, 141.497, 80.438, 7.528]
  MoveL 10055 to (-39.5, 155.15, 144.49) mm, rotated rx -180 ry 0 rz 180 deg; joints [-142.127, 74.047, -86.195, 141.497, 80.438, 7.528]
  Call Extruder(398.66562)
  MoveL 10056 to (-39.56, 154.97, 144.49) mm, rotated rx 180 ry 0 rz 180 deg; joints [-142.169, 74.042, -86.2, 141.538, 80.425, 7.527]
  MoveL 10057 to (-39.56, 154.97, 144.49) mm, rotated rx 180 ry 0 rz 180 deg; joints [-142.169, 74.042, -86.2, 141.538, 80.425, 7.527]
  Call Extruder(398.77796)
  MoveL 10058 to (-39.62, 154.78, 144.49) mm, rotated rx -180 ry 0 rz -180 deg; joints [-142.212, 74.038, -86.204, 141.58, 80.413, 7.525]
  MoveL 10059 to (-39.62, 154.78, 144.49) mm, rotated rx -180 ry 0 rz -180 deg; joints [-142.212, 74.038, -86.204, 141.58, 80.413, 7.525]
  Call Extruder(398.88986)
  MoveL 10060 to (-39.68, 154.59, 144.49) mm, rotated rx -180 ry 0 rz -180 deg; joints [-142.254, 74.033, -86.209, 141.621, 80.4, 7.524]
  MoveL 10061 to (-39.68, 154.59, 144.49) mm, rotated rx -180 ry 0 rz -180 deg; joints [-142.254, 74.033, -86.209, 141.621, 80.4, 7.524]
  Call Extruder(399.01126)
  MoveL 10062 to (-39.75, 154.38, 144.49) mm, rotated rx 180 ry 0 rz 180 deg; joints [-142.3, 74.029, -86.214, 141.666, 80.386, 7.523]
  MoveL 10063 to (-39.75, 154.38, 144.49) mm, rotated rx 180 ry 0 rz 180 deg; joints [-142.3, 74.029, -86.214, 141.666, 80.386, 7.523]
  Call Extruder(399.14206)
  MoveL 10064 to (-39.81, 154.16, 144.49) mm, rotated rx 180 ry 0 rz 180 deg; joints [-142.35, 74.023, -86.219, 141.715, 80.371, 7.521]
  MoveL 10065 to (-39.81, 154.16, 144.49) mm, rotated rx 180 ry 0 rz 180 deg; joints [-142.35, 74.023, -86.219, 141.715, 80.371, 7.521]
  Call Extruder(399.27229)
  MoveL 10066 to (-39.88, 153.94, 144.49) mm, rotated rx -180 ry 0 rz 180 deg; joints [-142.399, 74.017, -86.225, 141.764, 80.356, 7.52]
  MoveL 10067 to (-39.88, 153.94, 144.49) mm, rotated rx -180 ry 0 rz 180 deg; joints [-142.399, 74.017, -86.225, 141.764, 80.356, 7.52]
  Call Extruder(399.40195)
  MoveL 10068 to (-39.95, 153.71, 144.49) mm, rotated rx -180 ry 0 rz 180 deg; joints [-142.449, 74.012, -86.231, 141.812, 80.341, 7.518]
  MoveL 10069 to (-39.95, 153.71, 144.49) mm, rotated rx -180 ry 0 rz 180 deg; joints [-142.449, 74.012, -86.231, 141.812, 80.341, 7.518]
  Call Extruder(399.53105)
  MoveL 10070 to (-40.02, 153.49, 144.49) mm, rotated rx -180 ry 0 rz -180 deg; joints [-142.498, 74.006, -86.236, 141.861, 80.325, 7.517]
  MoveL 10071 to (-40.02, 153.49, 144.49) mm, rotated rx -180 ry 0 rz -180 deg; joints [-142.498, 74.006, -86.236, 141.861, 80.325, 7.517]
  Call Extruder(399.64614)
  MoveL 10072 to (-40.06, 153.28, 144.49) mm, rotated rx -180 ry 0 rz 180 deg; joints [-142.541, 74.001, -86.242, 141.903, 80.31, 7.517]
  MoveL 10073 to (-40.06, 153.28, 144.49) mm, rotated rx -180 ry 0 rz 180 deg; joints [-142.541, 74.001, -86.242, 141.903, 80.31, 7.517]
  Call Extruder(399.76077)
  MoveL 10074 to (-40.11, 153.08, 144.49) mm, rotated rx 180 ry 0 rz 180 deg; joints [-142.584, 73.995, -86.248, 141.945, 80.295, 7.517]
  MoveL 10075 to (-40.11, 153.08, 144.49) mm, rotated rx 180 ry 0 rz 180 deg; joints [-142.584, 73.995, -86.248, 141.945, 80.295, 7.517]
  Call Extruder(399.87495)
  MoveL 10076 to (-40.15, 152.88, 144.49) mm, rotated rx -180 ry 0 rz -180 deg; joints [-142.627, 73.989, -86.254, 141.987, 80.28, 7.518]
  MoveL 10077 to (-40.15, 152.88, 144.49) mm, rotated rx -180 ry 0 rz -180 deg; joints [-142.627, 73.989, -86.254, 141.987, 80.28, 7.518]
  Call Extruder(399.98868)
  MoveL 10078 to (-40.2, 152.67, 144.49) mm, rotated rx -180 ry 0 rz 180 deg; joints [-142.671, 73.983, -86.26, 142.029, 80.265, 7.518]
